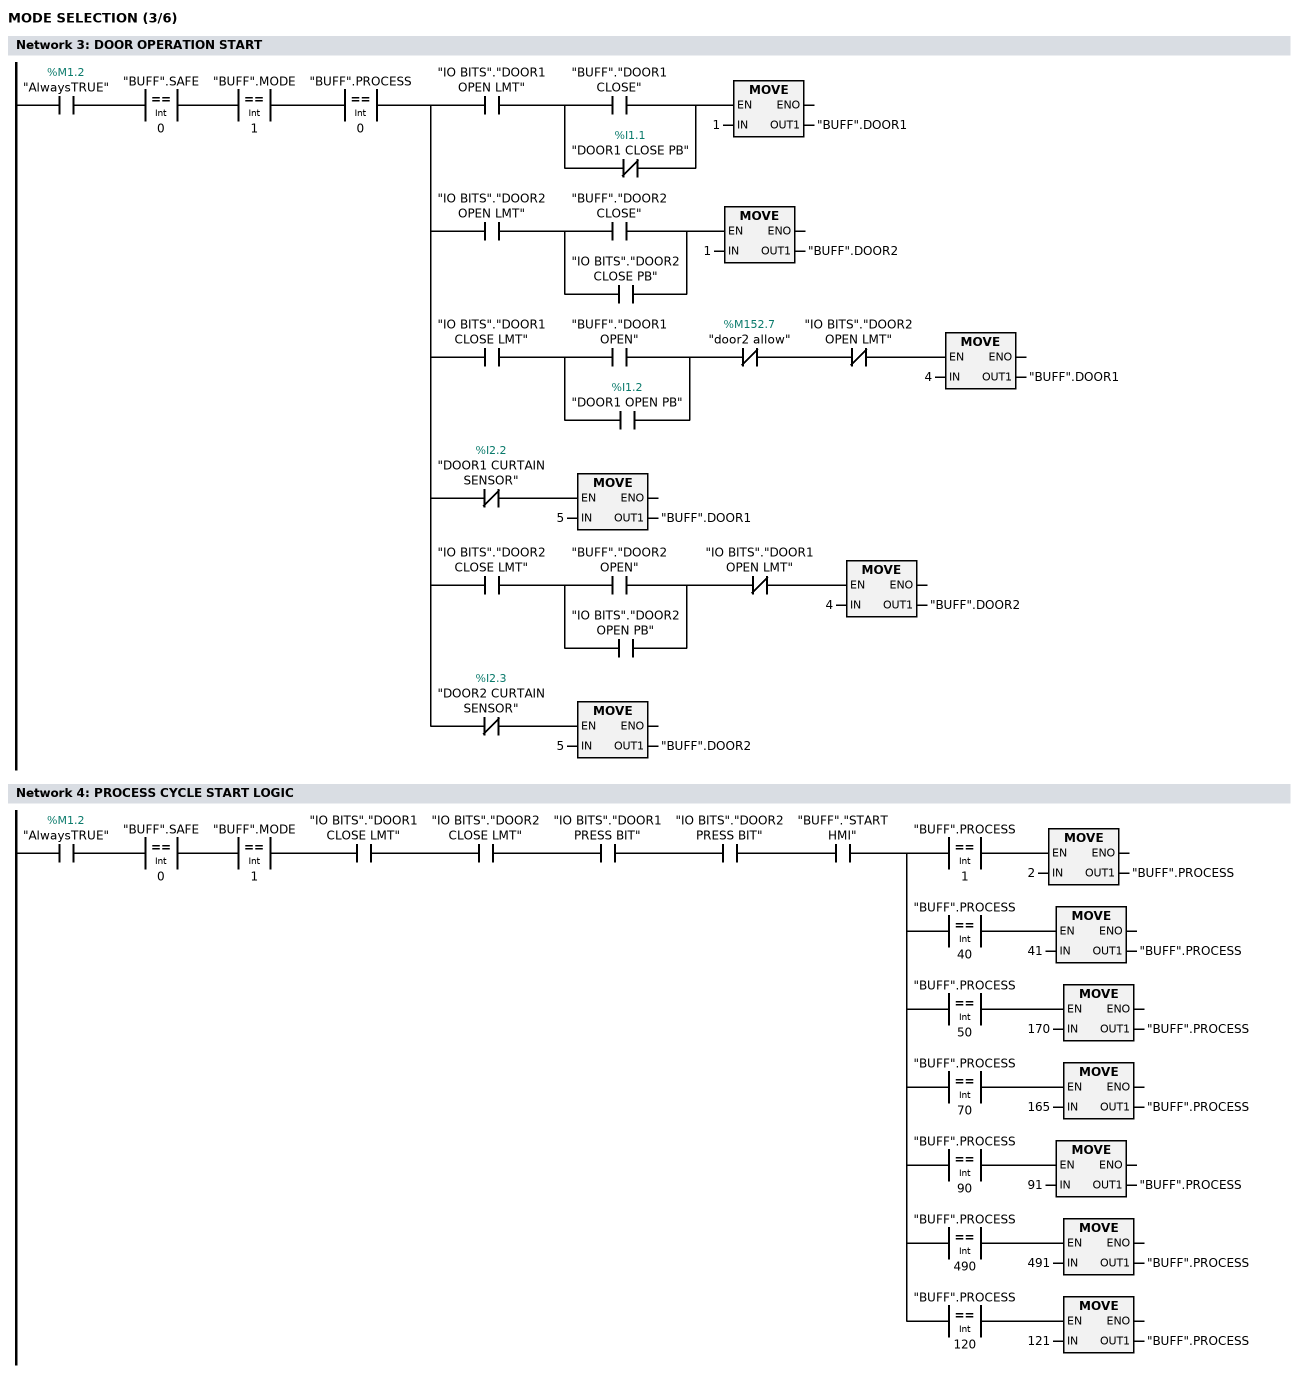
   RUNG wire#powerrail
      Contact( "AlwaysTRUE" )
      { S7_Templates := "SrcType := Int" } EQ_Contact(in1 := "BUFF".SAFE, in2 := 0)
      { S7_Templates := "SrcType := Int" } EQ_Contact(in1 := "BUFF".MODE, in2 := 1)
      { S7_Templates := "SrcType := Int" } EQ_Contact(in1 := "BUFF".PROCESS, in2 := 0)
      wire#w1
      Contact( "IO BITS"."DOOR1 OPEN LMT" )
      wire#w2
      Contact( "BUFF"."DOOR1 CLOSE" )
      wire#w3
      Move(in := 1, out1 => "BUFF".DOOR1)
   END_RUNG
   RUNG wire#w2
      I_Contact( "DOOR1 CLOSE PB" )
   END_RUNG wire#w3
   RUNG wire#w1
      Contact( "IO BITS"."DOOR2 OPEN LMT" )
      wire#w4
      Contact( "BUFF"."DOOR2 CLOSE" )
      wire#w5
      Move(in := 1, out1 => "BUFF".DOOR2)
   END_RUNG
   RUNG wire#w4
      Contact( "IO BITS"."DOOR2 CLOSE PB" )
   END_RUNG wire#w5
   RUNG wire#w1
      Contact( "IO BITS"."DOOR1 CLOSE LMT" )
      wire#w6
      Contact( "BUFF"."DOOR1 OPEN" )
      wire#w7
      I_Contact( "door2 allow" )
      I_Contact( "IO BITS"."DOOR2 OPEN LMT" )
      Move(in := 4, out1 => "BUFF".DOOR1)
   END_RUNG
   RUNG wire#w6
      Contact( "DOOR1 OPEN PB" )
   END_RUNG wire#w7
   RUNG wire#w1
      I_Contact( "DOOR1 CURTAIN SENSOR" )
      Move(in := 5, out1 => "BUFF".DOOR1)
   END_RUNG
   RUNG wire#w1
      Contact( "IO BITS"."DOOR2 CLOSE LMT" )
      wire#w8
      Contact( "BUFF"."DOOR2 OPEN" )
      wire#w9
      I_Contact( "IO BITS"."DOOR1 OPEN LMT" )
      Move(in := 4, out1 => "BUFF".DOOR2)
   END_RUNG
   RUNG wire#w8
      Contact( "IO BITS"."DOOR2 OPEN PB" )
   END_RUNG wire#w9
   RUNG wire#w1
      I_Contact( "DOOR2 CURTAIN SENSOR" )
      Move(in := 5, out1 => "BUFF".DOOR2)
   END_RUNG
   // the same network as SCL:
   #_w1 := "AlwaysTRUE" AND ("BUFF".SAFE = 0) AND ("BUFF".MODE = 1) AND ("BUFF".PROCESS = 0);
   IF #_w1 AND "IO BITS"."DOOR1 OPEN LMT" AND ("BUFF"."DOOR1 CLOSE" OR NOT "DOOR1 CLOSE PB") THEN
       "BUFF".DOOR1 := 1;
   END_IF;
   IF #_w1 AND "IO BITS"."DOOR2 OPEN LMT" AND ("BUFF"."DOOR2 CLOSE" OR "IO BITS"."DOOR2 CLOSE PB") THEN
       "BUFF".DOOR2 := 1;
   END_IF;
   IF #_w1 AND "IO BITS"."DOOR1 CLOSE LMT" AND ("BUFF"."DOOR1 OPEN" OR "DOOR1 OPEN PB") AND NOT "door2 allow" AND NOT "IO BITS"."DOOR2 OPEN LMT" THEN
       "BUFF".DOOR1 := 4;
   END_IF;
   IF #_w1 AND NOT "DOOR1 CURTAIN SENSOR" THEN "BUFF".DOOR1 := 5; END_IF;
   IF #_w1 AND "IO BITS"."DOOR2 CLOSE LMT" AND ("BUFF"."DOOR2 OPEN" OR "IO BITS"."DOOR2 OPEN PB") AND NOT "IO BITS"."DOOR1 OPEN LMT" THEN
       "BUFF".DOOR2 := 4;
   END_IF;
   IF #_w1 AND NOT "DOOR2 CURTAIN SENSOR" THEN "BUFF".DOOR2 := 5; END_IF;
END_REGION

REGION Network 4: PROCESS CYCLE START LOGIC
   RUNG wire#powerrail
      Contact( "AlwaysTRUE" )
      { S7_Templates := "SrcType := Int" } EQ_Contact(in1 := "BUFF".SAFE, in2 := 0)
      { S7_Templates := "SrcType := Int" } EQ_Contact(in1 := "BUFF".MODE, in2 := 1)
      Contact( "IO BITS"."DOOR1 CLOSE LMT" )
      Contact( "IO BITS"."DOOR2 CLOSE LMT" )
      Contact( "IO BITS"."DOOR1 PRESS BIT" )
      Contact( "IO BITS"."DOOR2 PRESS BIT" )
      Contact( "BUFF"."START HMI" )
      wire#w1
      { S7_Templates := "SrcType := Int" } EQ_Contact(in1 := "BUFF".PROCESS, in2 := 1)
      Move(in := 2, out1 => "BUFF".PROCESS)
   END_RUNG
   RUNG wire#w1
      { S7_Templates := "SrcType := Int" } EQ_Contact(in1 := "BUFF".PROCESS, in2 := 40)
      Move(in := 41, out1 => "BUFF".PROCESS)
   END_RUNG
   RUNG wire#w1
      { S7_Templates := "SrcType := Int" } EQ_Contact(in1 := "BUFF".PROCESS, in2 := 50)
      Move(in := 170, out1 => "BUFF".PROCESS)
   END_RUNG
   RUNG wire#w1
      { S7_Templates := "SrcType := Int" } EQ_Contact(in1 := "BUFF".PROCESS, in2 := 70)
      Move(in := 165, out1 => "BUFF".PROCESS)
   END_RUNG
   RUNG wire#w1
      { S7_Templates := "SrcType := Int" } EQ_Contact(in1 := "BUFF".PROCESS, in2 := 90)
      Move(in := 91, out1 => "BUFF".PROCESS)
   END_RUNG
   RUNG wire#w1
      { S7_Templates := "SrcType := Int" } EQ_Contact(in1 := "BUFF".PROCESS, in2 := 490)
      Move(in := 491, out1 => "BUFF".PROCESS)
   END_RUNG
   RUNG wire#w1
      { S7_Templates := "SrcType := Int" } EQ_Contact(in1 := "BUFF".PROCESS, in2 := 120)
      Move(in := 121, out1 => "BUFF".PROCESS)
   END_RUNG
   // the same network as SCL:
   #_w1 := "AlwaysTRUE" AND ("BUFF".SAFE = 0) AND ("BUFF".MODE = 1) AND "IO BITS"."DOOR1 CLOSE LMT" AND "IO BITS"."DOOR2 CLOSE LMT" AND "IO BITS"."DOOR1 PRESS BIT" AND "IO BITS"."DOOR2 PRESS BIT" AND "BUFF"."START HMI";
   IF #_w1 AND ("BUFF".PROCESS = 1) THEN "BUFF".PROCESS := 2; END_IF;
   IF #_w1 AND ("BUFF".PROCESS = 40) THEN "BUFF".PROCESS := 41; END_IF;
   IF #_w1 AND ("BUFF".PROCESS = 50) THEN "BUFF".PROCESS := 170; END_IF;
   IF #_w1 AND ("BUFF".PROCESS = 70) THEN "BUFF".PROCESS := 165; END_IF;
   IF #_w1 AND ("BUFF".PROCESS = 90) THEN "BUFF".PROCESS := 91; END_IF;
   IF #_w1 AND ("BUFF".PROCESS = 490) THEN "BUFF".PROCESS := 491; END_IF;
   IF #_w1 AND ("BUFF".PROCESS = 120) THEN "BUFF".PROCESS := 121; END_IF;
END_REGION

REGION Network 5: DOOR CLOSE LOGIC
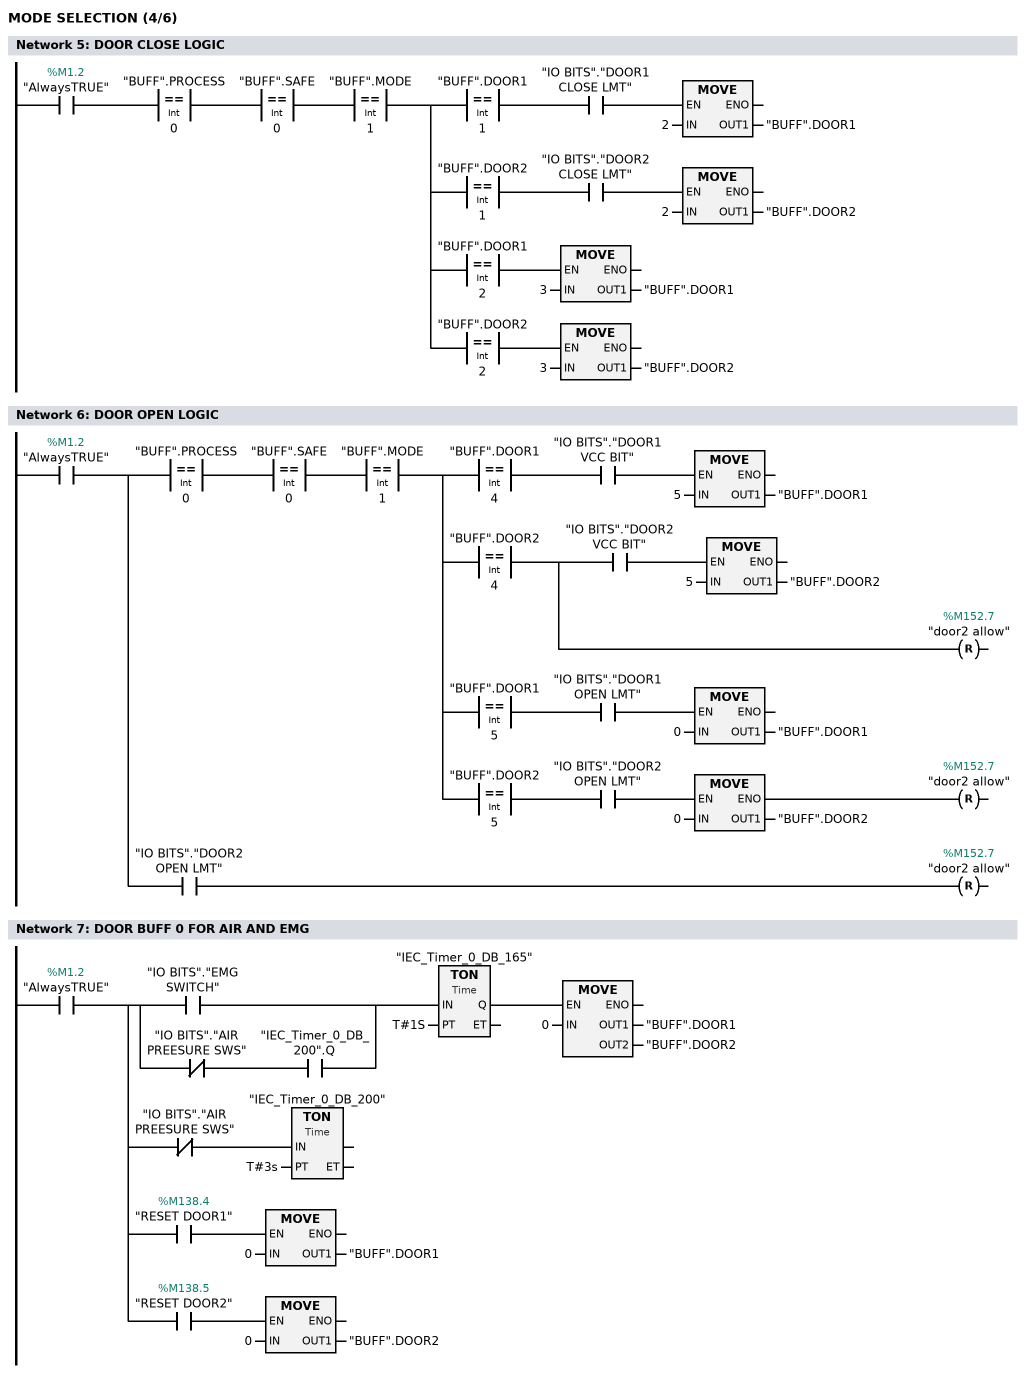
   RUNG wire#powerrail
      Contact( "AlwaysTRUE" )
      { S7_Templates := "SrcType := Int" } EQ_Contact(in1 := "BUFF".PROCESS, in2 := 0)
      { S7_Templates := "SrcType := Int" } EQ_Contact(in1 := "BUFF".SAFE, in2 := 0)
      { S7_Templates := "SrcType := Int" } EQ_Contact(in1 := "BUFF".MODE, in2 := 1)
      wire#w1
      { S7_Templates := "SrcType := Int" } EQ_Contact(in1 := "BUFF".DOOR1, in2 := 1)
      Contact( "IO BITS"."DOOR1 CLOSE LMT" )
      Move(in := 2, out1 => "BUFF".DOOR1)
   END_RUNG
   RUNG wire#w1
      { S7_Templates := "SrcType := Int" } EQ_Contact(in1 := "BUFF".DOOR2, in2 := 1)
      Contact( "IO BITS"."DOOR2 CLOSE LMT" )
      Move(in := 2, out1 => "BUFF".DOOR2)
   END_RUNG
   RUNG wire#w1
      { S7_Templates := "SrcType := Int" } EQ_Contact(in1 := "BUFF".DOOR1, in2 := 2)
      Move(in := 3, out1 => "BUFF".DOOR1)
   END_RUNG
   RUNG wire#w1
      { S7_Templates := "SrcType := Int" } EQ_Contact(in1 := "BUFF".DOOR2, in2 := 2)
      Move(in := 3, out1 => "BUFF".DOOR2)
   END_RUNG
   // the same network as SCL:
   #_w1 := "AlwaysTRUE" AND ("BUFF".PROCESS = 0) AND ("BUFF".SAFE = 0) AND ("BUFF".MODE = 1);
   IF #_w1 AND ("BUFF".DOOR1 = 1) AND "IO BITS"."DOOR1 CLOSE LMT" THEN "BUFF".DOOR1 := 2; END_IF;
   IF #_w1 AND ("BUFF".DOOR2 = 1) AND "IO BITS"."DOOR2 CLOSE LMT" THEN "BUFF".DOOR2 := 2; END_IF;
   IF #_w1 AND ("BUFF".DOOR1 = 2) THEN "BUFF".DOOR1 := 3; END_IF;
   IF #_w1 AND ("BUFF".DOOR2 = 2) THEN "BUFF".DOOR2 := 3; END_IF;
END_REGION

REGION Network 6: DOOR OPEN LOGIC
   RUNG wire#powerrail
      Contact( "AlwaysTRUE" )
      wire#w1
      { S7_Templates := "SrcType := Int" } EQ_Contact(in1 := "BUFF".PROCESS, in2 := 0)
      { S7_Templates := "SrcType := Int" } EQ_Contact(in1 := "BUFF".SAFE, in2 := 0)
      { S7_Templates := "SrcType := Int" } EQ_Contact(in1 := "BUFF".MODE, in2 := 1)
      wire#w2
      { S7_Templates := "SrcType := Int" } EQ_Contact(in1 := "BUFF".DOOR1, in2 := 4)
      Contact( "IO BITS"."DOOR1 VCC BIT" )
      Move(in := 5, out1 => "BUFF".DOOR1)
   END_RUNG
   RUNG wire#w2
      { S7_Templates := "SrcType := Int" } EQ_Contact(in1 := "BUFF".DOOR2, in2 := 4)
      wire#w3
      Contact( "IO BITS"."DOOR2 VCC BIT" )
      Move(in := 5, out1 => "BUFF".DOOR2)
   END_RUNG
   RUNG wire#w3
      R_Coil( "door2 allow" )
   END_RUNG
   RUNG wire#w2
      { S7_Templates := "SrcType := Int" } EQ_Contact(in1 := "BUFF".DOOR1, in2 := 5)
      Contact( "IO BITS"."DOOR1 OPEN LMT" )
      Move(in := 0, out1 => "BUFF".DOOR1)
   END_RUNG
   RUNG wire#w2
      { S7_Templates := "SrcType := Int" } EQ_Contact(in1 := "BUFF".DOOR2, in2 := 5)
      Contact( "IO BITS"."DOOR2 OPEN LMT" )
      Move(in := 0, out1 => "BUFF".DOOR2)
      R_Coil( "door2 allow" )
   END_RUNG
   RUNG wire#w1
      Contact( "IO BITS"."DOOR2 OPEN LMT" )
      R_Coil( "door2 allow" )
   END_RUNG
   // the same network as SCL:
   #_w1 := "AlwaysTRUE" AND ("BUFF".PROCESS = 0) AND ("BUFF".SAFE = 0) AND ("BUFF".MODE = 1);
   IF #_w1 AND ("BUFF".DOOR1 = 4) AND "IO BITS"."DOOR1 VCC BIT" THEN "BUFF".DOOR1 := 5; END_IF;
   #_w2 := #_w1 AND ("BUFF".DOOR2 = 4);
   IF #_w2 AND "IO BITS"."DOOR2 VCC BIT" THEN "BUFF".DOOR2 := 5; END_IF;
   IF #_w2 THEN "door2 allow" := FALSE; END_IF;
   IF #_w1 AND ("BUFF".DOOR1 = 5) AND "IO BITS"."DOOR1 OPEN LMT" THEN "BUFF".DOOR1 := 0; END_IF;
   #_w3 := #_w1 AND ("BUFF".DOOR2 = 5) AND "IO BITS"."DOOR2 OPEN LMT";
   IF #_w3 THEN
       "BUFF".DOOR2 := 0;
       "door2 allow" := FALSE;
   END_IF;
   IF "AlwaysTRUE" AND "IO BITS"."DOOR2 OPEN LMT" THEN "door2 allow" := FALSE; END_IF;
END_REGION

REGION Network 7: DOOR BUFF 0 FOR AIR AND EMG
   RUNG wire#powerrail
      Contact( "AlwaysTRUE" )
      wire#w1
      Contact( "IO BITS"."EMG SWITCH" )
      wire#w2
      { S7_Templates := "time_type := Time" } "IEC_Timer_0_DB_165".TON(pt := T#1S, et =>)
      Move(in := 0, out1 => "BUFF".DOOR1, out2 => "BUFF".DOOR2)
   END_RUNG
   RUNG wire#w1
      I_Contact( "IO BITS"."AIR PREESURE SWS" )
      Contact( "IEC_Timer_0_DB_200".Q )
   END_RUNG wire#w2
   RUNG wire#w1
      I_Contact( "IO BITS"."AIR PREESURE SWS" )
      { S7_Templates := "time_type := Time" } "IEC_Timer_0_DB_200".TON(pt := T#3s, et =>)
   END_RUNG
   RUNG wire#w1
      Contact( "RESET DOOR1" )
      Move(in := 0, out1 => "BUFF".DOOR1)
   END_RUNG
   RUNG wire#w1
      Contact( "RESET DOOR2" )
      Move(in := 0, out1 => "BUFF".DOOR2)
   END_RUNG
   // the same network as SCL:
   "IEC_Timer_0_DB_165".TON(IN := "AlwaysTRUE" AND ("IO BITS"."EMG SWITCH" OR (NOT "IO BITS"."AIR PREESURE SWS" AND "IEC_Timer_0_DB_200".Q)),
                           PT := T#1S);
   IF "IEC_Timer_0_DB_165".Q THEN
       "BUFF".DOOR1 := 0;
       "BUFF".DOOR2 := 0;
   END_IF;
   "IEC_Timer_0_DB_200".TON(IN := "AlwaysTRUE" AND NOT "IO BITS"."AIR PREESURE SWS", PT := T#3s);
   IF "AlwaysTRUE" AND "RESET DOOR1" THEN "BUFF".DOOR1 := 0; END_IF;
   IF "AlwaysTRUE" AND "RESET DOOR2" THEN "BUFF".DOOR2 := 0; END_IF;
END_REGION

REGION Network 8: MANUAL RESET
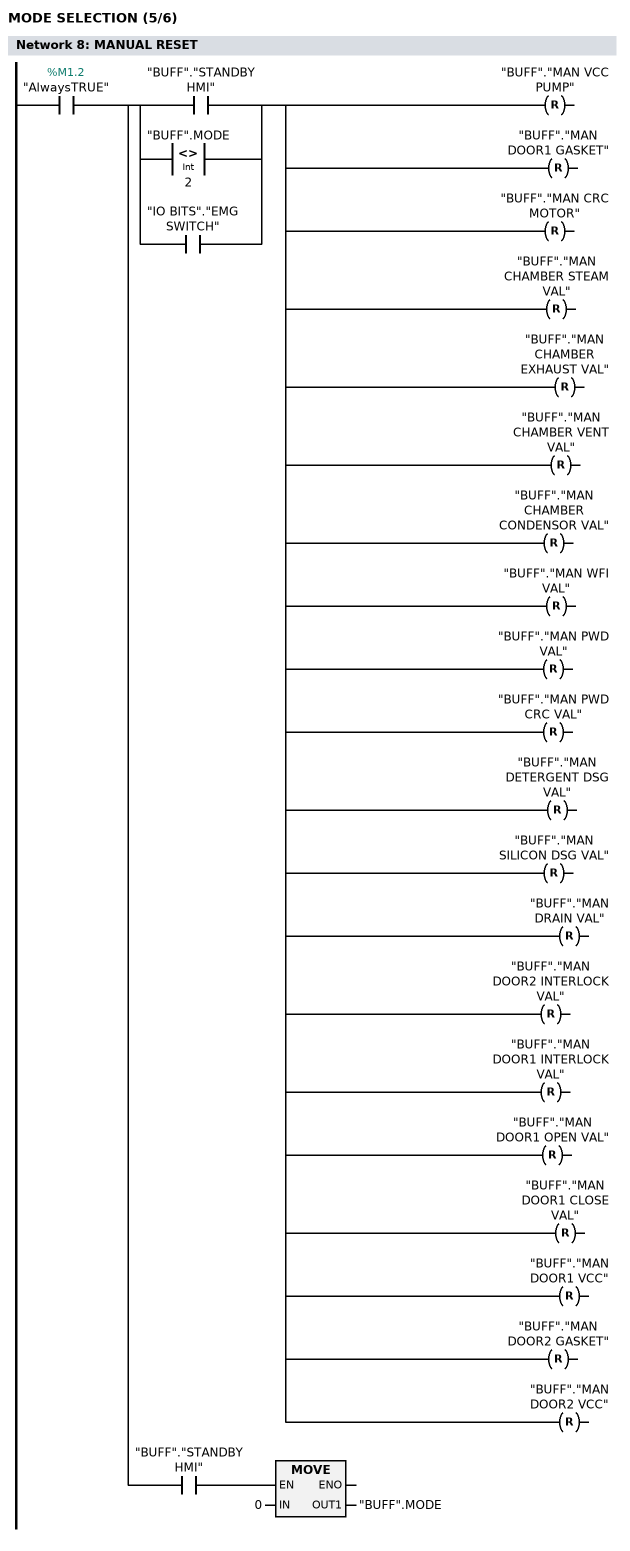
   RUNG wire#powerrail
      Contact( "AlwaysTRUE" )
      wire#w1
      Contact( "BUFF"."STANDBY HMI" )
      wire#w2
      R_Coil( "BUFF"."MAN VCC PUMP" )
   END_RUNG
   RUNG wire#w1
      { S7_Templates := "SrcType := Int" } NE_Contact(in1 := "BUFF".MODE, in2 := 2)
   END_RUNG wire#w2
   RUNG wire#w1
      Contact( "IO BITS"."EMG SWITCH" )
   END_RUNG wire#w2
   RUNG wire#w2
      R_Coil( "BUFF"."MAN DOOR1 GASKET" )
   END_RUNG
   RUNG wire#w2
      R_Coil( "BUFF"."MAN CRC MOTOR" )
   END_RUNG
   RUNG wire#w2
      R_Coil( "BUFF"."MAN CHAMBER STEAM VAL" )
   END_RUNG
   RUNG wire#w2
      R_Coil( "BUFF"."MAN CHAMBER EXHAUST VAL" )
   END_RUNG
   RUNG wire#w2
      R_Coil( "BUFF"."MAN CHAMBER VENT VAL" )
   END_RUNG
   RUNG wire#w2
      R_Coil( "BUFF"."MAN CHAMBER CONDENSOR VAL" )
   END_RUNG
   RUNG wire#w2
      R_Coil( "BUFF"."MAN WFI VAL" )
   END_RUNG
   RUNG wire#w2
      R_Coil( "BUFF"."MAN PWD VAL" )
   END_RUNG
   RUNG wire#w2
      R_Coil( "BUFF"."MAN PWD CRC VAL" )
   END_RUNG
   RUNG wire#w2
      R_Coil( "BUFF"."MAN DETERGENT DSG VAL" )
   END_RUNG
   RUNG wire#w2
      R_Coil( "BUFF"."MAN SILICON DSG VAL" )
   END_RUNG
   RUNG wire#w2
      R_Coil( "BUFF"."MAN DRAIN VAL" )
   END_RUNG
   RUNG wire#w2
      R_Coil( "BUFF"."MAN DOOR2 INTERLOCK VAL" )
   END_RUNG
   RUNG wire#w2
      R_Coil( "BUFF"."MAN DOOR1 INTERLOCK VAL" )
   END_RUNG
   RUNG wire#w2
      R_Coil( "BUFF"."MAN DOOR1 OPEN VAL" )
   END_RUNG
   RUNG wire#w2
      R_Coil( "BUFF"."MAN DOOR1 CLOSE VAL" )
   END_RUNG
   RUNG wire#w2
      R_Coil( "BUFF"."MAN DOOR1 VCC" )
   END_RUNG
   RUNG wire#w2
      R_Coil( "BUFF"."MAN DOOR2 GASKET" )
   END_RUNG
   RUNG wire#w2
      R_Coil( "BUFF"."MAN DOOR2 VCC" )
   END_RUNG
   RUNG wire#w1
      Contact( "BUFF"."STANDBY HMI" )
      Move(in := 0, out1 => "BUFF".MODE)
   END_RUNG
   // the same network as SCL:
   IF "AlwaysTRUE" AND ("BUFF"."STANDBY HMI" OR ("BUFF".MODE <> 2) OR "IO BITS"."EMG SWITCH") THEN
       "BUFF"."MAN VCC PUMP" := FALSE;
       "BUFF"."MAN DOOR1 GASKET" := FALSE;
       "BUFF"."MAN CRC MOTOR" := FALSE;
       "BUFF"."MAN CHAMBER STEAM VAL" := FALSE;
       "BUFF"."MAN CHAMBER EXHAUST VAL" := FALSE;
       "BUFF"."MAN CHAMBER VENT VAL" := FALSE;
       "BUFF"."MAN CHAMBER CONDENSOR VAL" := FALSE;
       "BUFF"."MAN WFI VAL" := FALSE;
       "BUFF"."MAN PWD VAL" := FALSE;
       "BUFF"."MAN PWD CRC VAL" := FALSE;
       "BUFF"."MAN DETERGENT DSG VAL" := FALSE;
       "BUFF"."MAN SILICON DSG VAL" := FALSE;
       "BUFF"."MAN DRAIN VAL" := FALSE;
       "BUFF"."MAN DOOR2 INTERLOCK VAL" := FALSE;
       "BUFF"."MAN DOOR1 INTERLOCK VAL" := FALSE;
       "BUFF"."MAN DOOR1 OPEN VAL" := FALSE;
       "BUFF"."MAN DOOR1 CLOSE VAL" := FALSE;
       "BUFF"."MAN DOOR1 VCC" := FALSE;
       "BUFF"."MAN DOOR2 GASKET" := FALSE;
       "BUFF"."MAN DOOR2 VCC" := FALSE;
   END_IF;
   IF "AlwaysTRUE" AND "BUFF"."STANDBY HMI" THEN "BUFF".MODE := 0; END_IF;
END_REGION

REGION Network 9
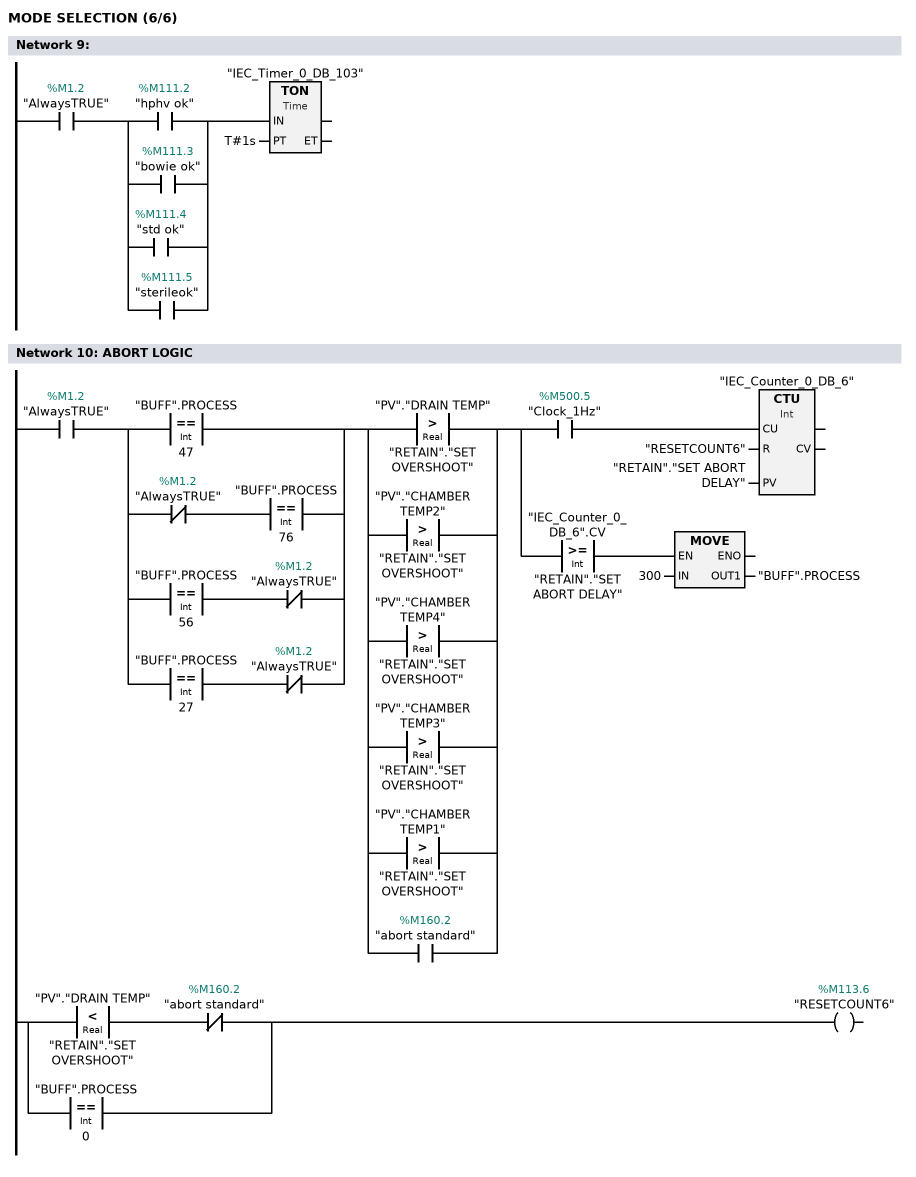
   RUNG wire#powerrail
      Contact( "AlwaysTRUE" )
      wire#w1
      Contact( "hphv ok" )
      wire#w2
      { S7_Templates := "time_type := Time" } "IEC_Timer_0_DB_103".TON(pt := T#1s, et =>)
   END_RUNG
   RUNG wire#w1
      Contact( "bowie ok" )
   END_RUNG wire#w2
   RUNG wire#w1
      Contact( "std ok" )
   END_RUNG wire#w2
   RUNG wire#w1
      Contact( "sterileok" )
   END_RUNG wire#w2
   // the same network as SCL:
   "IEC_Timer_0_DB_103".TON(IN := "AlwaysTRUE" AND ("hphv ok" OR "bowie ok" OR "std ok" OR "sterileok"),
                           PT := T#1s);
END_REGION

REGION Network 10: ABORT LOGIC
   RUNG wire#powerrail
      Contact( "AlwaysTRUE" )
      wire#w1
      { S7_Templates := "SrcType := Int" } EQ_Contact(in1 := "BUFF".PROCESS, in2 := 47)
      wire#w2
      { S7_Templates := "SrcType := Real" } GT_Contact(in1 := "PV"."DRAIN TEMP", in2 := "RETAIN"."SET OVERSHOOT")
      wire#w3
      Contact( "Clock_1Hz" )
      { S7_Templates := "value_type := Int" } "IEC_Counter_0_DB_6".CTU(r := "RESETCOUNT6", pv := "RETAIN"."SET ABORT DELAY", cv =>)
   END_RUNG
   RUNG wire#w1
      I_Contact( "AlwaysTRUE" )
      { S7_Templates := "SrcType := Int" } EQ_Contact(in1 := "BUFF".PROCESS, in2 := 76)
   END_RUNG wire#w2
   RUNG wire#w1
      { S7_Templates := "SrcType := Int" } EQ_Contact(in1 := "BUFF".PROCESS, in2 := 56)
      I_Contact( "AlwaysTRUE" )
   END_RUNG wire#w2
   RUNG wire#w1
      { S7_Templates := "SrcType := Int" } EQ_Contact(in1 := "BUFF".PROCESS, in2 := 27)
      I_Contact( "AlwaysTRUE" )
   END_RUNG wire#w2
   RUNG wire#w2
      { S7_Templates := "SrcType := Real" } GT_Contact(in1 := "PV"."CHAMBER TEMP2", in2 := "RETAIN"."SET OVERSHOOT")
   END_RUNG wire#w3
   RUNG wire#w2
      { S7_Templates := "SrcType := Real" } GT_Contact(in1 := "PV"."CHAMBER TEMP4", in2 := "RETAIN"."SET OVERSHOOT")
   END_RUNG wire#w3
   RUNG wire#w2
      { S7_Templates := "SrcType := Real" } GT_Contact(in1 := "PV"."CHAMBER TEMP3", in2 := "RETAIN"."SET OVERSHOOT")
   END_RUNG wire#w3
   RUNG wire#w2
      { S7_Templates := "SrcType := Real" } GT_Contact(in1 := "PV"."CHAMBER TEMP1", in2 := "RETAIN"."SET OVERSHOOT")
   END_RUNG wire#w3
   RUNG wire#w2
      Contact( "abort standard" )
   END_RUNG wire#w3
   RUNG wire#w3
      { S7_Templates := "SrcType := Int" } GE_Contact(in1 := "IEC_Counter_0_DB_6".CV, in2 := "RETAIN"."SET ABORT DELAY")
      Move(in := 300, out1 => "BUFF".PROCESS)
   END_RUNG
   RUNG wire#powerrail
      { S7_Templates := "SrcType := Real" } LT_Contact(in1 := "PV"."DRAIN TEMP", in2 := "RETAIN"."SET OVERSHOOT")
      I_Contact( "abort standard" )
      wire#w4
      Coil( "RESETCOUNT6" )
   END_RUNG
   RUNG wire#powerrail
      { S7_Templates := "SrcType := Int" } EQ_Contact(in1 := "BUFF".PROCESS, in2 := 0)
   END_RUNG wire#w4
   // the same network as SCL:
   #_w1 := "AlwaysTRUE" AND (("BUFF".PROCESS = 47) OR (NOT "AlwaysTRUE" AND ("BUFF".PROCESS = 76)) OR (("BUFF".PROCESS = 56) AND NOT "AlwaysTRUE") OR (("BUFF".PROCESS = 27) AND NOT "AlwaysTRUE")) AND (("PV"."DRAIN TEMP" > "RETAIN"."SET OVERSHOOT") OR ("PV"."CHAMBER TEMP2" > "RETAIN"."SET OVERSHOOT") OR ("PV"."CHAMBER TEMP4" > "RETAIN"."SET OVERSHOOT") OR ("PV"."CHAMBER TEMP3" > "RETAIN"."SET OVERSHOOT") OR ("PV"."CHAMBER TEMP1" > "RETAIN"."SET OVERSHOOT") OR "abort standard");
   "IEC_Counter_0_DB_6".CTU(CU := #_w1 AND "Clock_1Hz", R := "RESETCOUNT6", PV := "RETAIN"."SET ABORT DELAY");
   IF #_w1 AND ("IEC_Counter_0_DB_6".CV >= "RETAIN"."SET ABORT DELAY") THEN "BUFF".PROCESS := 300; END_IF;
   "RESETCOUNT6" := (("PV"."DRAIN TEMP" < "RETAIN"."SET OVERSHOOT") AND NOT "abort standard") OR ("BUFF".PROCESS = 0);
END_REGION
END_FUNCTION

FUNCTION "ANALOG" : Void   // FC9, LAD
{ S7_Optimized_Access := 'TRUE' }
// stored: SetENOAutomatically false
   VAR_TEMP
      DOOR1_P : Real;
      DOOR2_P : Real;
      CHAMBER_P : Real;
      JACKET_P : Real;
      NOM : Real;
      TEMP1 : Real;
   END_VAR
   VAR_TEMP   // added for the SCL form of the ladder/FBD networks
      _w1 : Bool;
      _w2 : Bool;
      _w3 : Bool;
   END_VAR
BEGIN

REGION Network 1: TEMPERATURE RTD
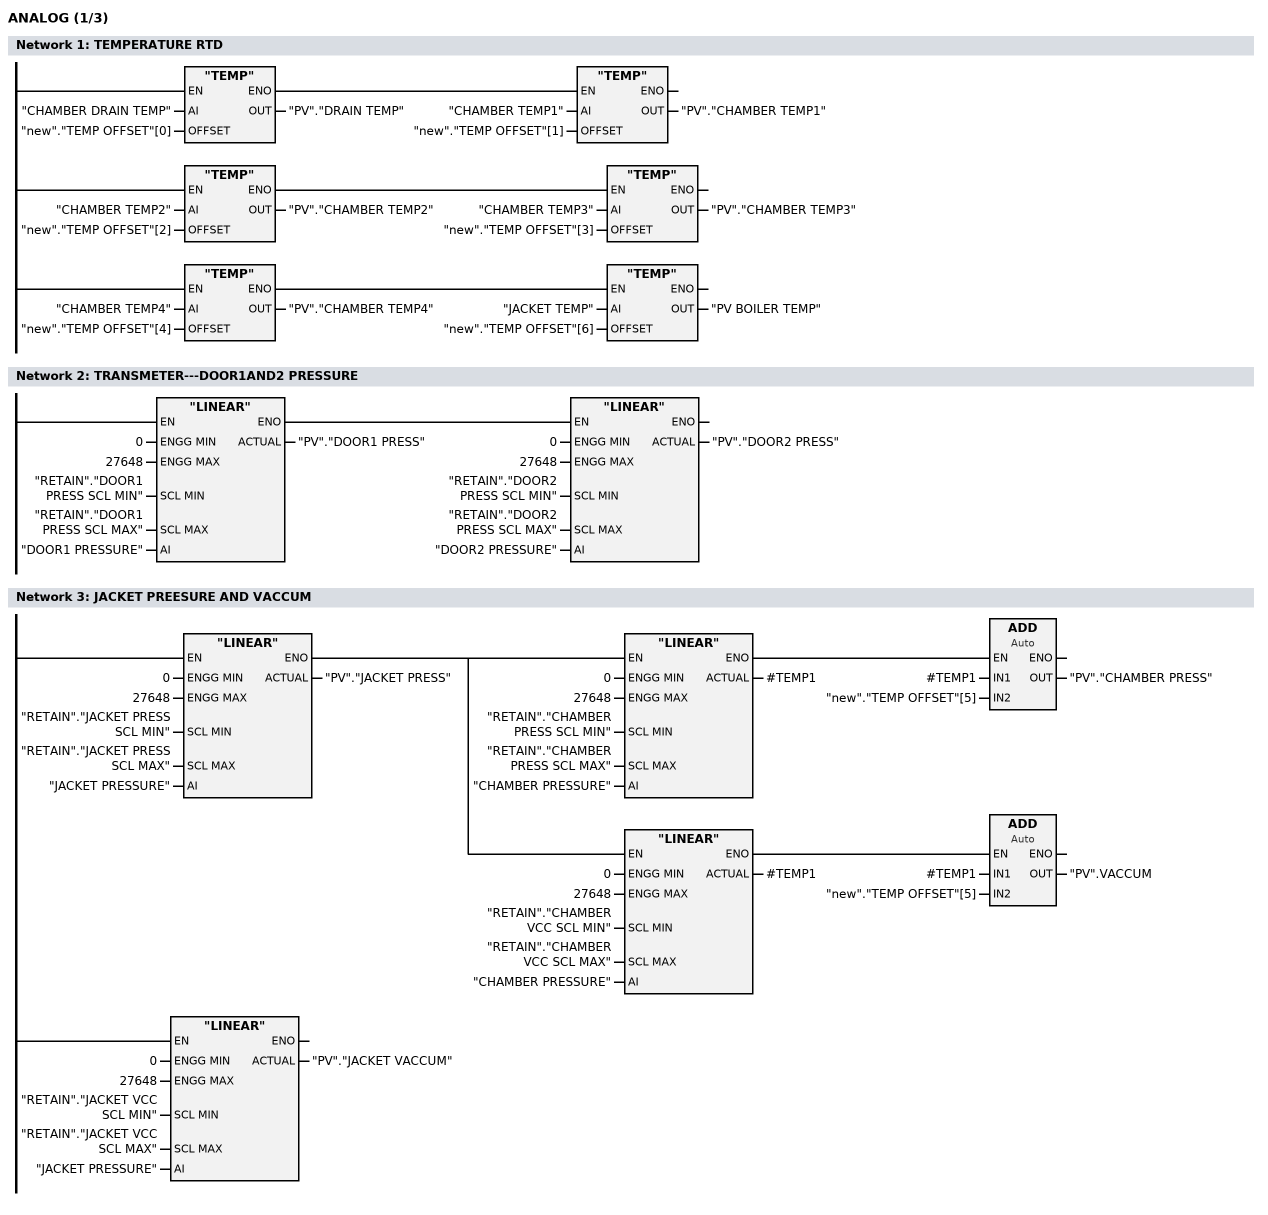
   RUNG wire#powerrail
      "TEMP"(AI := "CHAMBER DRAIN TEMP", OFFSET := "new"."TEMP OFFSET"[0], OUT => "PV"."DRAIN TEMP")
      "TEMP"(AI := "CHAMBER TEMP1", OFFSET := "new"."TEMP OFFSET"[1], OUT => "PV"."CHAMBER TEMP1")
   END_RUNG
   RUNG wire#powerrail
      "TEMP"(AI := "CHAMBER TEMP2", OFFSET := "new"."TEMP OFFSET"[2], OUT => "PV"."CHAMBER TEMP2")
      "TEMP"(AI := "CHAMBER TEMP3", OFFSET := "new"."TEMP OFFSET"[3], OUT => "PV"."CHAMBER TEMP3")
   END_RUNG
   RUNG wire#powerrail
      "TEMP"(AI := "CHAMBER TEMP4", OFFSET := "new"."TEMP OFFSET"[4], OUT => "PV"."CHAMBER TEMP4")
      "TEMP"(AI := "JACKET TEMP", OFFSET := "new"."TEMP OFFSET"[6], OUT => "PV BOILER TEMP")
   END_RUNG
   // the same network as SCL:
   "TEMP"(AI := "CHAMBER DRAIN TEMP", OFFSET := "new"."TEMP OFFSET"[0], OUT => "PV"."DRAIN TEMP", ENO => #_w1);
   IF #_w1 THEN
       "TEMP"(AI := "CHAMBER TEMP1", OFFSET := "new"."TEMP OFFSET"[1], OUT => "PV"."CHAMBER TEMP1");
   END_IF;
   "TEMP"(AI := "CHAMBER TEMP2", OFFSET := "new"."TEMP OFFSET"[2], OUT => "PV"."CHAMBER TEMP2", ENO => #_w2);
   IF #_w2 THEN
       "TEMP"(AI := "CHAMBER TEMP3", OFFSET := "new"."TEMP OFFSET"[3], OUT => "PV"."CHAMBER TEMP3");
   END_IF;
   "TEMP"(AI := "CHAMBER TEMP4", OFFSET := "new"."TEMP OFFSET"[4], OUT => "PV"."CHAMBER TEMP4", ENO => #_w3);
   IF #_w3 THEN
       "TEMP"(AI := "JACKET TEMP", OFFSET := "new"."TEMP OFFSET"[6], OUT => "PV BOILER TEMP");
   END_IF;
END_REGION

REGION Network 2: TRANSMETER---DOOR1AND2 PRESSURE
   RUNG wire#powerrail
      "LINEAR"("ENGG MIN" := 0, "ENGG MAX" := 27648, "SCL MIN" := "RETAIN"."DOOR1 PRESS SCL MIN", "SCL MAX" := "RETAIN"."DOOR1 PRESS SCL MAX", AI := "DOOR1 PRESSURE", ACTUAL => "PV"."DOOR1 PRESS")
      "LINEAR"("ENGG MIN" := 0, "ENGG MAX" := 27648, "SCL MIN" := "RETAIN"."DOOR2 PRESS SCL MIN", "SCL MAX" := "RETAIN"."DOOR2 PRESS SCL MAX", AI := "DOOR2 PRESSURE", ACTUAL => "PV"."DOOR2 PRESS")
   END_RUNG
   // the same network as SCL:
   "LINEAR"("ENGG MIN" := 0,
            "ENGG MAX" := 27648,
            "SCL MIN" := "RETAIN"."DOOR1 PRESS SCL MIN",
            "SCL MAX" := "RETAIN"."DOOR1 PRESS SCL MAX",
            AI := "DOOR1 PRESSURE",
            ACTUAL => "PV"."DOOR1 PRESS",
            ENO => #_w1);
   IF #_w1 THEN
       "LINEAR"("ENGG MIN" := 0,
                "ENGG MAX" := 27648,
                "SCL MIN" := "RETAIN"."DOOR2 PRESS SCL MIN",
                "SCL MAX" := "RETAIN"."DOOR2 PRESS SCL MAX",
                AI := "DOOR2 PRESSURE",
                ACTUAL => "PV"."DOOR2 PRESS");
   END_IF;
END_REGION

REGION Network 3: JACKET PREESURE AND VACCUM
   RUNG wire#powerrail
      "LINEAR"("ENGG MIN" := 0, "ENGG MAX" := 27648, "SCL MIN" := "RETAIN"."JACKET PRESS SCL MIN", "SCL MAX" := "RETAIN"."JACKET PRESS SCL MAX", AI := "JACKET PRESSURE", ACTUAL => "PV"."JACKET PRESS")
      wire#w1
      "LINEAR"("ENGG MIN" := 0, "ENGG MAX" := 27648, "SCL MIN" := "RETAIN"."CHAMBER PRESS SCL MIN", "SCL MAX" := "RETAIN"."CHAMBER PRESS SCL MAX", AI := "CHAMBER PRESSURE", ACTUAL => #TEMP1)
      Add(in1 := #TEMP1, in2 := "new"."TEMP OFFSET"[5], out => "PV"."CHAMBER PRESS")
   END_RUNG
   RUNG wire#w1
      "LINEAR"("ENGG MIN" := 0, "ENGG MAX" := 27648, "SCL MIN" := "RETAIN"."CHAMBER VCC SCL MIN", "SCL MAX" := "RETAIN"."CHAMBER VCC SCL MAX", AI := "CHAMBER PRESSURE", ACTUAL => #TEMP1)
      Add(in1 := #TEMP1, in2 := "new"."TEMP OFFSET"[5], out => "PV".VACCUM)
   END_RUNG
   RUNG wire#powerrail
      "LINEAR"("ENGG MIN" := 0, "ENGG MAX" := 27648, "SCL MIN" := "RETAIN"."JACKET VCC SCL MIN", "SCL MAX" := "RETAIN"."JACKET VCC SCL MAX", AI := "JACKET PRESSURE", ACTUAL => "PV"."JACKET VACCUM")
   END_RUNG
   // the same network as SCL:
   "LINEAR"("ENGG MIN" := 0,
            "ENGG MAX" := 27648,
            "SCL MIN" := "RETAIN"."JACKET PRESS SCL MIN",
            "SCL MAX" := "RETAIN"."JACKET PRESS SCL MAX",
            AI := "JACKET PRESSURE",
            ACTUAL => "PV"."JACKET PRESS",
            ENO => #_w1);
   "LINEAR"(EN := #_w1,
            "ENGG MIN" := 0,
            "ENGG MAX" := 27648,
            "SCL MIN" := "RETAIN"."CHAMBER PRESS SCL MIN",
            "SCL MAX" := "RETAIN"."CHAMBER PRESS SCL MAX",
            AI := "CHAMBER PRESSURE",
            ACTUAL => #TEMP1,
            ENO => #_w2);
   IF #_w2 THEN "PV"."CHAMBER PRESS" := #TEMP1 + "new"."TEMP OFFSET"[5]; END_IF;
   "LINEAR"(EN := #_w1,
            "ENGG MIN" := 0,
            "ENGG MAX" := 27648,
            "SCL MIN" := "RETAIN"."CHAMBER VCC SCL MIN",
            "SCL MAX" := "RETAIN"."CHAMBER VCC SCL MAX",
            AI := "CHAMBER PRESSURE",
            ACTUAL => #TEMP1,
            ENO => #_w3);
   IF #_w3 THEN "PV".VACCUM := #TEMP1 + "new"."TEMP OFFSET"[5]; END_IF;
   "LINEAR"("ENGG MIN" := 0,
            "ENGG MAX" := 27648,
            "SCL MIN" := "RETAIN"."JACKET VCC SCL MIN",
            "SCL MAX" := "RETAIN"."JACKET VCC SCL MAX",
            AI := "JACKET PRESSURE",
            ACTUAL => "PV"."JACKET VACCUM");
END_REGION

REGION Network 4: DOOR1AND 2 VACCUM
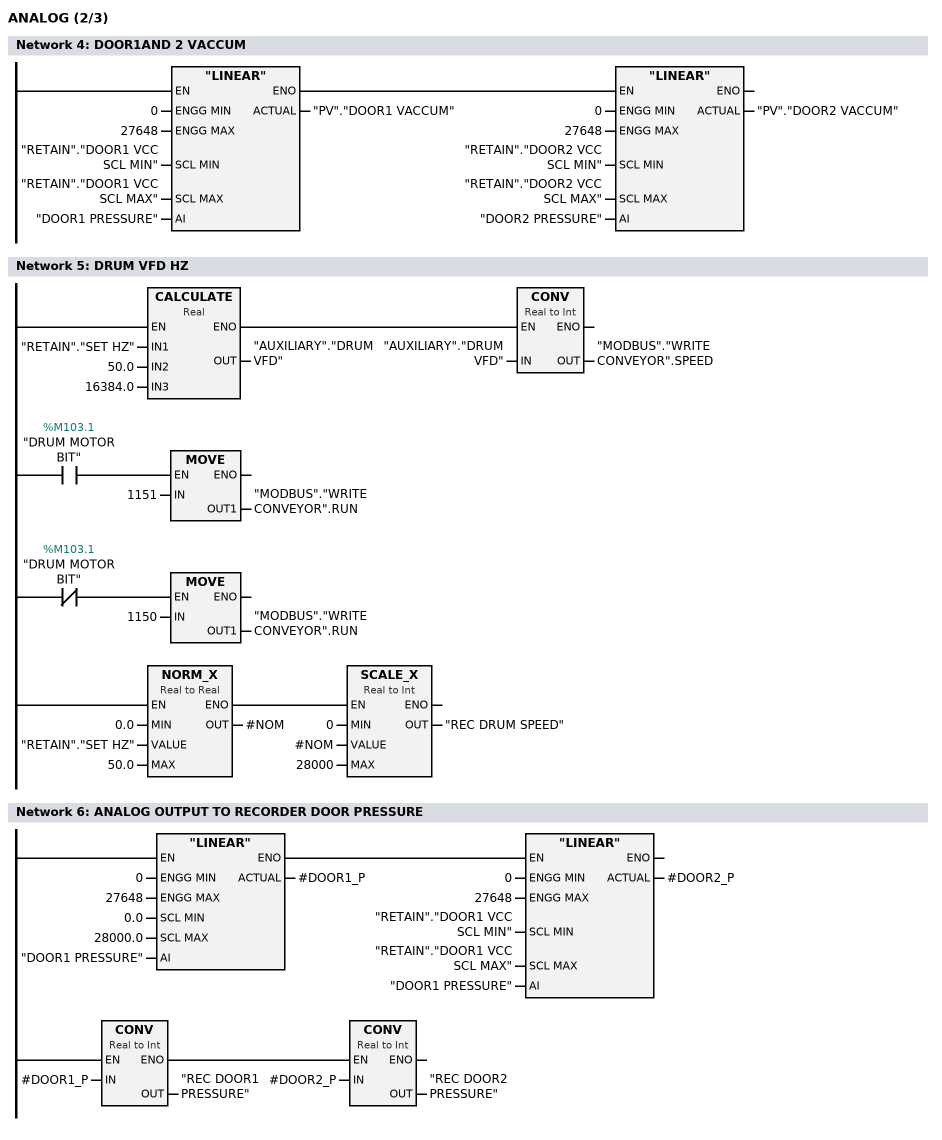
   RUNG wire#powerrail
      "LINEAR"("ENGG MIN" := 0, "ENGG MAX" := 27648, "SCL MIN" := "RETAIN"."DOOR1 VCC SCL MIN", "SCL MAX" := "RETAIN"."DOOR1 VCC SCL MAX", AI := "DOOR1 PRESSURE", ACTUAL => "PV"."DOOR1 VACCUM")
      "LINEAR"("ENGG MIN" := 0, "ENGG MAX" := 27648, "SCL MIN" := "RETAIN"."DOOR2 VCC SCL MIN", "SCL MAX" := "RETAIN"."DOOR2 VCC SCL MAX", AI := "DOOR2 PRESSURE", ACTUAL => "PV"."DOOR2 VACCUM")
   END_RUNG
   // the same network as SCL:
   "LINEAR"("ENGG MIN" := 0,
            "ENGG MAX" := 27648,
            "SCL MIN" := "RETAIN"."DOOR1 VCC SCL MIN",
            "SCL MAX" := "RETAIN"."DOOR1 VCC SCL MAX",
            AI := "DOOR1 PRESSURE",
            ACTUAL => "PV"."DOOR1 VACCUM",
            ENO => #_w1);
   IF #_w1 THEN
       "LINEAR"("ENGG MIN" := 0,
                "ENGG MAX" := 27648,
                "SCL MIN" := "RETAIN"."DOOR2 VCC SCL MIN",
                "SCL MAX" := "RETAIN"."DOOR2 VCC SCL MAX",
                AI := "DOOR2 PRESSURE",
                ACTUAL => "PV"."DOOR2 VACCUM");
   END_IF;
END_REGION

REGION Network 5: DRUM VFD HZ
   RUNG wire#powerrail
      { S7_Templates := "SrcType := Real"; S7_Expression := "(IN1/IN2)*IN3" } Calculate(in1 := "RETAIN"."SET HZ", in2 := 50.0, in3 := 16384.0, out => "AUXILIARY"."DRUM VFD")
      { S7_Templates := "[SrcType := Real, DestType := Int]" } Convert(in := "AUXILIARY"."DRUM VFD", out => "MODBUS"."WRITE CONVEYOR".SPEED)
   END_RUNG
   RUNG wire#powerrail
      Contact( "DRUM MOTOR BIT" )
      Move(in := 1151, out1 => "MODBUS"."WRITE CONVEYOR".RUN)
   END_RUNG
   RUNG wire#powerrail
      I_Contact( "DRUM MOTOR BIT" )
      Move(in := 1150, out1 => "MODBUS"."WRITE CONVEYOR".RUN)
   END_RUNG
   RUNG wire#powerrail
      { S7_Templates := "[SrcType := Real, DestType := Real]" } Normalize(min := 0.0, value := "RETAIN"."SET HZ", max := 50.0, out => #NOM)
      { S7_Templates := "[SrcType := Real, DestType := Int]" } Scale(min := 0, value := #NOM, max := 28000, out => "REC DRUM SPEED")
   END_RUNG
   // the same network as SCL:
   "AUXILIARY"."DRUM VFD" := ("RETAIN"."SET HZ"/50.0)*16384.0;
   "MODBUS"."WRITE CONVEYOR".SPEED := REAL_TO_INT("AUXILIARY"."DRUM VFD");
   IF "DRUM MOTOR BIT" THEN "MODBUS"."WRITE CONVEYOR".RUN := 1151; END_IF;
   IF NOT "DRUM MOTOR BIT" THEN "MODBUS"."WRITE CONVEYOR".RUN := 1150; END_IF;
   #NOM := NORM_X(MIN := 0.0, VALUE := "RETAIN"."SET HZ", MAX := 50.0);
   "REC DRUM SPEED" := SCALE_X(MIN := 0, VALUE := #NOM, MAX := 28000);
END_REGION

REGION Network 6: ANALOG OUTPUT TO RECORDER DOOR PRESSURE
   RUNG wire#powerrail
      "LINEAR"("ENGG MIN" := 0, "ENGG MAX" := 27648, "SCL MIN" := 0.0, "SCL MAX" := 28000.0, AI := "DOOR1 PRESSURE", ACTUAL => #DOOR1_P)
      "LINEAR"("ENGG MIN" := 0, "ENGG MAX" := 27648, "SCL MIN" := "RETAIN"."DOOR1 VCC SCL MIN", "SCL MAX" := "RETAIN"."DOOR1 VCC SCL MAX", AI := "DOOR1 PRESSURE", ACTUAL => #DOOR2_P)
   END_RUNG
   RUNG wire#powerrail
      { S7_Templates := "[SrcType := Real, DestType := Int]" } Convert(in := #DOOR1_P, out => "REC DOOR1 PRESSURE")
      { S7_Templates := "[SrcType := Real, DestType := Int]" } Convert(in := #DOOR2_P, out => "REC DOOR2 PRESSURE")
   END_RUNG
   // the same network as SCL:
   "LINEAR"("ENGG MIN" := 0,
            "ENGG MAX" := 27648,
            "SCL MIN" := 0.0,
            "SCL MAX" := 28000.0,
            AI := "DOOR1 PRESSURE",
            ACTUAL => #DOOR1_P,
            ENO => #_w1);
   IF #_w1 THEN
       "LINEAR"("ENGG MIN" := 0,
                "ENGG MAX" := 27648,
                "SCL MIN" := "RETAIN"."DOOR1 VCC SCL MIN",
                "SCL MAX" := "RETAIN"."DOOR1 VCC SCL MAX",
                AI := "DOOR1 PRESSURE",
                ACTUAL => #DOOR2_P);
   END_IF;
   "REC DOOR1 PRESSURE" := REAL_TO_INT(#DOOR1_P);
   "REC DOOR2 PRESSURE" := REAL_TO_INT(#DOOR2_P);
END_REGION

REGION Network 7: ANALOG OUTPUT TO RECORDER CHAMBER AND JACKET
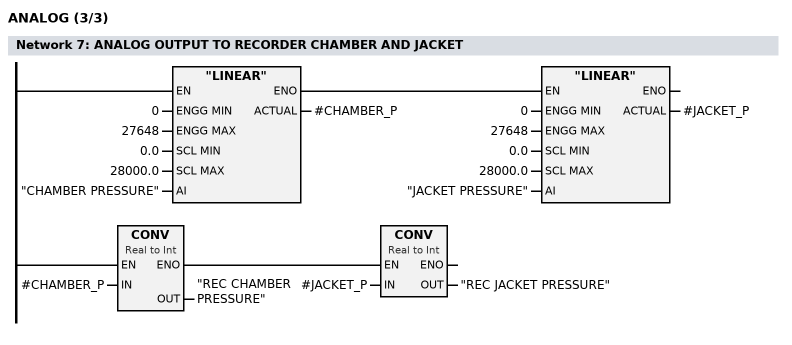
   RUNG wire#powerrail
      "LINEAR"("ENGG MIN" := 0, "ENGG MAX" := 27648, "SCL MIN" := 0.0, "SCL MAX" := 28000.0, AI := "CHAMBER PRESSURE", ACTUAL => #CHAMBER_P)
      "LINEAR"("ENGG MIN" := 0, "ENGG MAX" := 27648, "SCL MIN" := 0.0, "SCL MAX" := 28000.0, AI := "JACKET PRESSURE", ACTUAL => #JACKET_P)
   END_RUNG
   RUNG wire#powerrail
      { S7_Templates := "[SrcType := Real, DestType := Int]" } Convert(in := #CHAMBER_P, out => "REC CHAMBER PRESSURE")
      { S7_Templates := "[SrcType := Real, DestType := Int]" } Convert(in := #JACKET_P, out => "REC JACKET PRESSURE")
   END_RUNG
   // the same network as SCL:
   "LINEAR"("ENGG MIN" := 0,
            "ENGG MAX" := 27648,
            "SCL MIN" := 0.0,
            "SCL MAX" := 28000.0,
            AI := "CHAMBER PRESSURE",
            ACTUAL => #CHAMBER_P,
            ENO => #_w1);
   IF #_w1 THEN
       "LINEAR"("ENGG MIN" := 0,
                "ENGG MAX" := 27648,
                "SCL MIN" := 0.0,
                "SCL MAX" := 28000.0,
                AI := "JACKET PRESSURE",
                ACTUAL => #JACKET_P);
   END_IF;
   "REC CHAMBER PRESSURE" := REAL_TO_INT(#CHAMBER_P);
   "REC JACKET PRESSURE" := REAL_TO_INT(#JACKET_P);
END_REGION
END_FUNCTION

FUNCTION "TEMP" : Void   // FC14, LAD
{ S7_Optimized_Access := 'TRUE' }
// stored: SetENOAutomatically false
   VAR_INPUT
      AI : Int;
      OFFSET : Real;
   END_VAR
   VAR_OUTPUT
      OUT : Real;
   END_VAR
   VAR_TEMP
      TEMP1 : Real;
      temp2 : Real;
   END_VAR
BEGIN

REGION Network 1
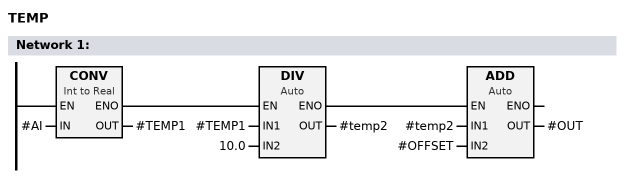
   RUNG wire#powerrail
      { S7_Templates := "[SrcType := Int, DestType := Real]" } Convert(in := #AI, out => #TEMP1)
      Div(in1 := #TEMP1, in2 := 10.0, out => #temp2)
      Add(in1 := #temp2, in2 := #OFFSET, out => #OUT)
   END_RUNG
   // the same network as SCL:
   #TEMP1 := INT_TO_REAL(#AI);
   #temp2 := #TEMP1 / 10.0;
   #OUT := #temp2 + #OFFSET;
END_REGION
END_FUNCTION

FUNCTION "LINEAR" : Void   // FC15, LAD
{ S7_Optimized_Access := 'TRUE' }
// stored: SetENOAutomatically false
   VAR_INPUT
      "ENGG MIN" : Int;
      "ENGG MAX" : Int;
      "SCL MIN" : Real;
      "SCL MAX" : Real;
      AI : Int;
   END_VAR
   VAR_OUTPUT
      ACTUAL : Real;
   END_VAR
   VAR_TEMP
      NOM : Real;
   END_VAR
BEGIN

REGION Network 1
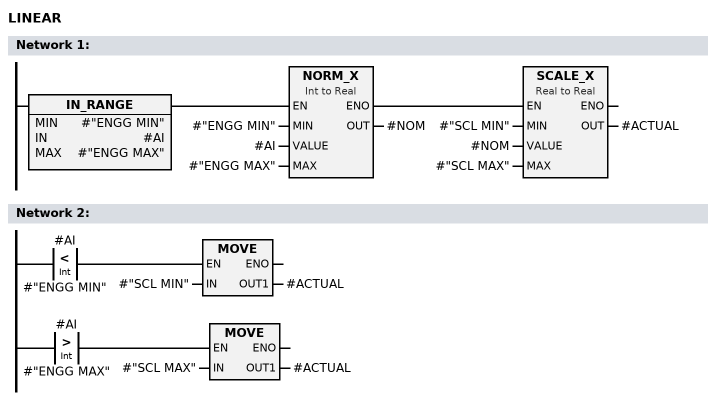
   RUNG wire#powerrail
      { S7_Templates := "SrcType := Int" } InRange(min := #"ENGG MIN", in := #AI, max := #"ENGG MAX")
      { S7_Templates := "[SrcType := Int, DestType := Real]" } Normalize(min := #"ENGG MIN", value := #AI, max := #"ENGG MAX", out => #NOM)
      { S7_Templates := "[SrcType := Real, DestType := Real]" } Scale(min := #"SCL MIN", value := #NOM, max := #"SCL MAX", out => #ACTUAL)
   END_RUNG
   // the same network as SCL:
   IF (#"ENGG MIN" <= #AI) AND (#AI <= #"ENGG MAX") THEN
       #NOM := NORM_X(MIN := #"ENGG MIN", VALUE := #AI, MAX := #"ENGG MAX");
       #ACTUAL := SCALE_X(MIN := #"SCL MIN", VALUE := #NOM, MAX := #"SCL MAX");
   END_IF;
END_REGION

REGION Network 2
   RUNG wire#powerrail
      { S7_Templates := "SrcType := Int" } LT_Contact(in1 := #AI, in2 := #"ENGG MIN")
      Move(in := #"SCL MIN", out1 => #ACTUAL)
   END_RUNG
   RUNG wire#powerrail
      { S7_Templates := "SrcType := Int" } GT_Contact(in1 := #AI, in2 := #"ENGG MAX")
      Move(in := #"SCL MAX", out1 => #ACTUAL)
   END_RUNG
   // the same network as SCL:
   IF #AI < #"ENGG MIN" THEN #ACTUAL := #"SCL MIN"; END_IF;
   IF #AI > #"ENGG MAX" THEN #ACTUAL := #"SCL MAX"; END_IF;
END_REGION
END_FUNCTION

FUNCTION "DELTA" : Void   // FC18, LAD
{ S7_Optimized_Access := 'TRUE' }
// stored: SetENOAutomatically false
   VAR_TEMP
      "F1 VALUE" : Real;
      "F2 VALUE" : Real;
      "F3 VALUE" : Real;
      "F4 VALUE" : Real;
      "F5 VALUE" : Real;
   END_VAR
   VAR_TEMP   // added for the SCL form of the ladder/FBD networks
      _w1 : Bool;
      _w2 : Bool;
      _w3 : Bool;
      _w4 : Bool;
      _w5 : Bool;
      _w6 : Bool;
      _w7 : Bool;
      _w8 : Bool;
      _w9 : Bool;
      _w10 : Bool;
      _w11 : Bool;
      _w12 : Bool;
   END_VAR
BEGIN

REGION Network 1
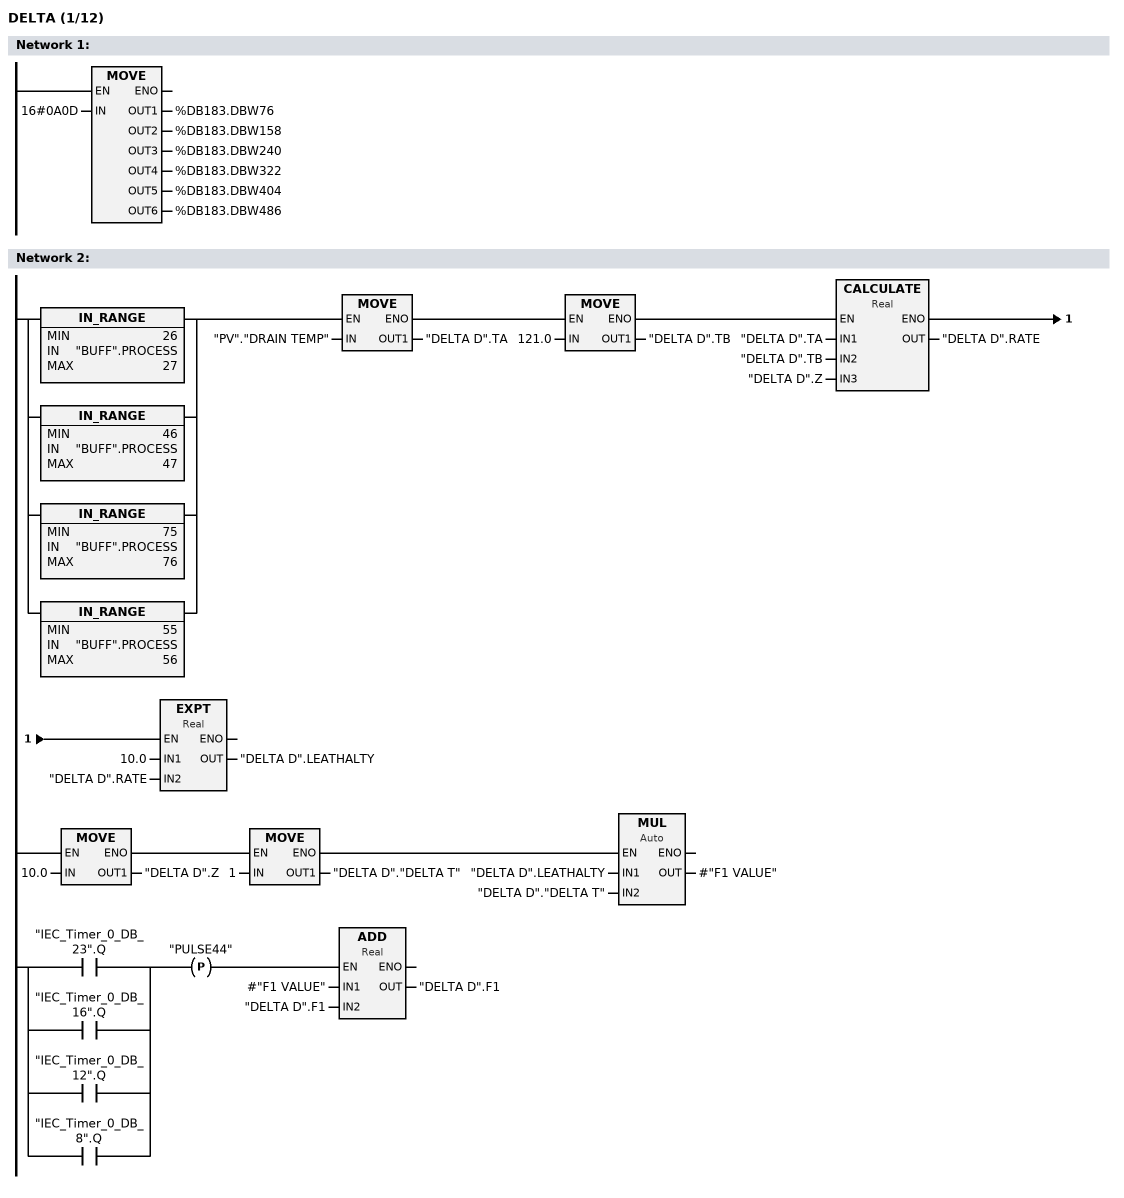
   RUNG wire#powerrail
      Move(in := 16#0A0D, out1 => %DB183.DBW76, out2 => %DB183.DBW158, out3 => %DB183.DBW240, out4 => %DB183.DBW322, out5 => %DB183.DBW404, out6 => %DB183.DBW486)
   END_RUNG
   // the same network as SCL:
   %DB183.DBW76 := 16#0A0D;
   %DB183.DBW158 := 16#0A0D;
   %DB183.DBW240 := 16#0A0D;
   %DB183.DBW322 := 16#0A0D;
   %DB183.DBW404 := 16#0A0D;
   %DB183.DBW486 := 16#0A0D;
END_REGION

REGION Network 2
   IF ((26 <= "BUFF".PROCESS) AND ("BUFF".PROCESS <= 27)) OR ((46 <= "BUFF".PROCESS) AND ("BUFF".PROCESS <= 47)) OR ((75 <= "BUFF".PROCESS) AND ("BUFF".PROCESS <= 76)) OR ((55 <= "BUFF".PROCESS) AND ("BUFF".PROCESS <= 56)) THEN
       "DELTA D".TA := "PV"."DRAIN TEMP";
       "DELTA D".TB := 121.0;
       "DELTA D".RATE := ("DELTA D".TA-"DELTA D".TB)/"DELTA D".Z;
       "DELTA D".LEATHALTY := 10.0 ** "DELTA D".RATE;
   END_IF;
   "DELTA D".Z := 10.0;
   "DELTA D"."DELTA T" := 1;
   #"F1 VALUE" := "DELTA D".LEATHALTY * "DELTA D"."DELTA T";
   #_w1 := "IEC_Timer_0_DB_23".Q OR "IEC_Timer_0_DB_16".Q OR "IEC_Timer_0_DB_12".Q OR "IEC_Timer_0_DB_8".Q;
   #_w2 := #_w1 AND NOT "PULSE44";   // rising edge
   "PULSE44" := #_w1;
   IF #_w2 THEN "DELTA D".F1 := #"F1 VALUE" + "DELTA D".F1; END_IF;
END_REGION

REGION Network 3
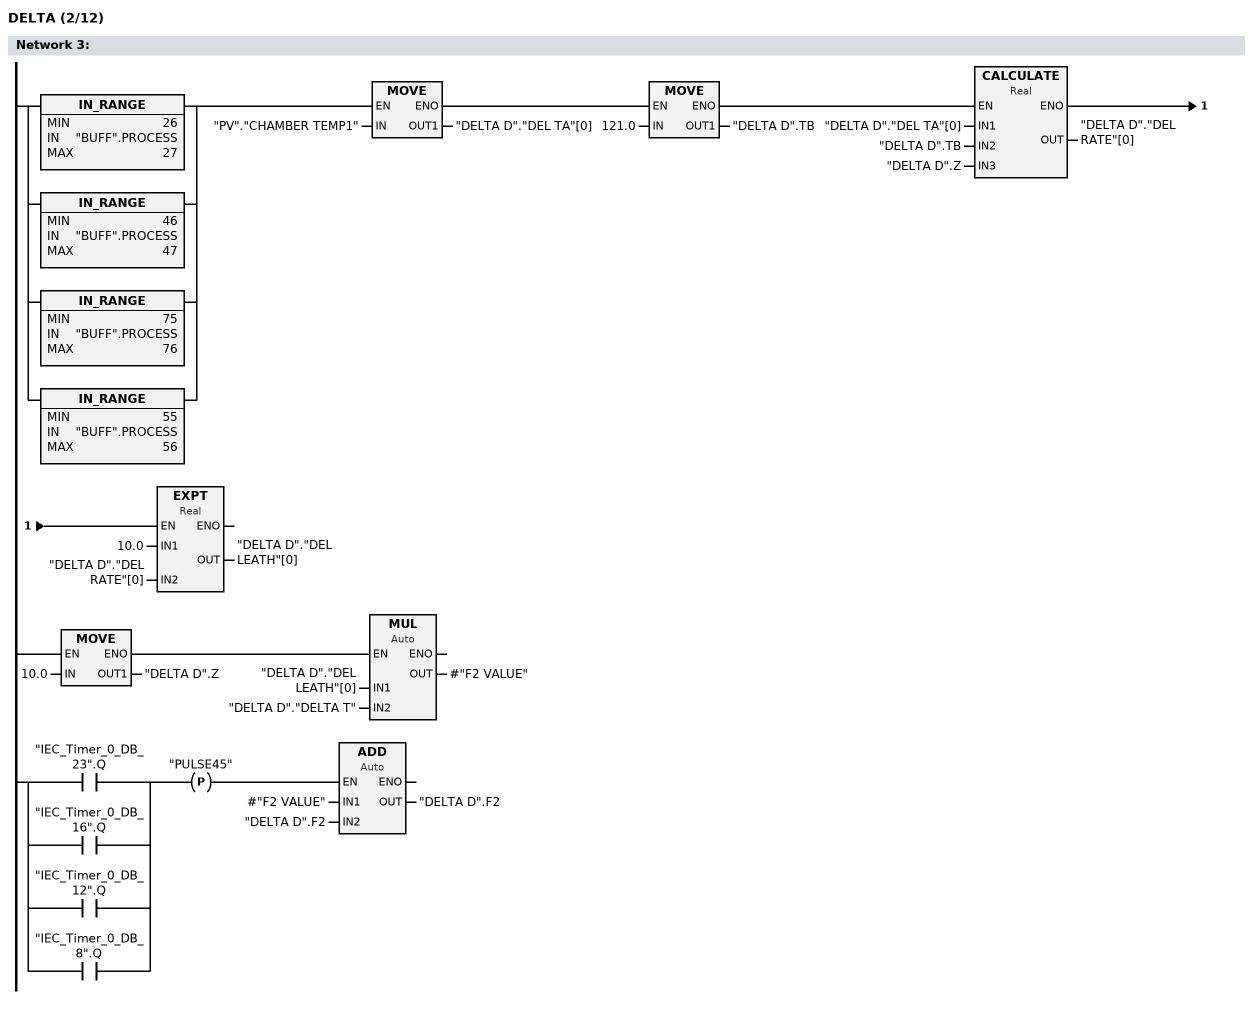
   IF ((26 <= "BUFF".PROCESS) AND ("BUFF".PROCESS <= 27)) OR ((46 <= "BUFF".PROCESS) AND ("BUFF".PROCESS <= 47)) OR ((75 <= "BUFF".PROCESS) AND ("BUFF".PROCESS <= 76)) OR ((55 <= "BUFF".PROCESS) AND ("BUFF".PROCESS <= 56)) THEN
       "DELTA D"."DEL TA"[0] := "PV"."CHAMBER TEMP1";
       "DELTA D".TB := 121.0;
       "DELTA D"."DEL RATE"[0] := ("DELTA D"."DEL TA"[0]-"DELTA D".TB)/"DELTA D".Z;
       "DELTA D"."DEL LEATH"[0] := 10.0 ** "DELTA D"."DEL RATE"[0];
   END_IF;
   "DELTA D".Z := 10.0;
   #"F2 VALUE" := "DELTA D"."DEL LEATH"[0] * "DELTA D"."DELTA T";
   #_w1 := "IEC_Timer_0_DB_23".Q OR "IEC_Timer_0_DB_16".Q OR "IEC_Timer_0_DB_12".Q OR "IEC_Timer_0_DB_8".Q;
   #_w2 := #_w1 AND NOT "PULSE45";   // rising edge
   "PULSE45" := #_w1;
   IF #_w2 THEN "DELTA D".F2 := #"F2 VALUE" + "DELTA D".F2; END_IF;
END_REGION

REGION Network 4
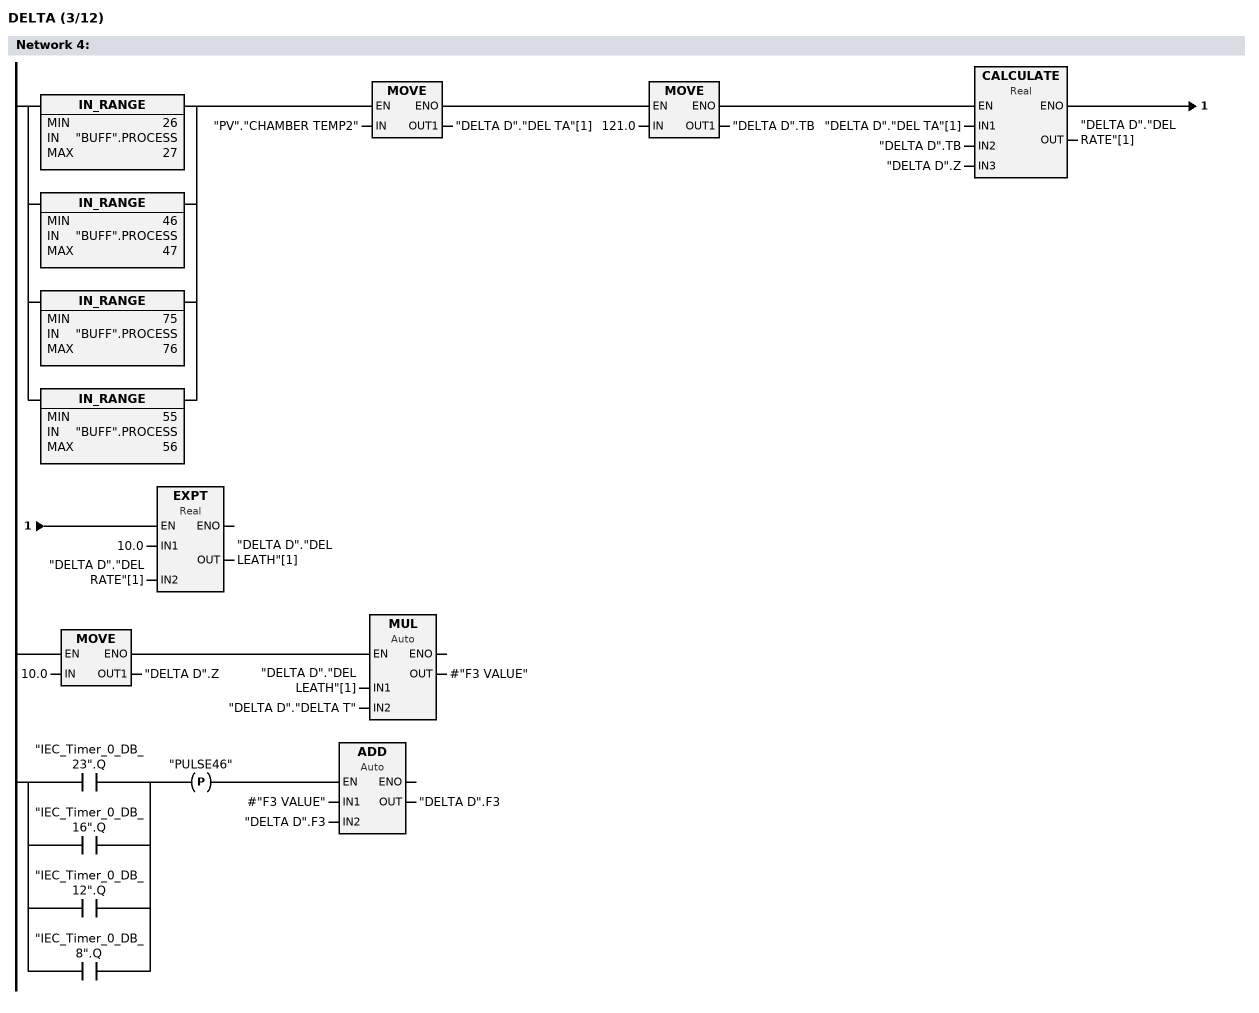
   IF ((26 <= "BUFF".PROCESS) AND ("BUFF".PROCESS <= 27)) OR ((46 <= "BUFF".PROCESS) AND ("BUFF".PROCESS <= 47)) OR ((75 <= "BUFF".PROCESS) AND ("BUFF".PROCESS <= 76)) OR ((55 <= "BUFF".PROCESS) AND ("BUFF".PROCESS <= 56)) THEN
       "DELTA D"."DEL TA"[1] := "PV"."CHAMBER TEMP2";
       "DELTA D".TB := 121.0;
       "DELTA D"."DEL RATE"[1] := ("DELTA D"."DEL TA"[1]-"DELTA D".TB)/"DELTA D".Z;
       "DELTA D"."DEL LEATH"[1] := 10.0 ** "DELTA D"."DEL RATE"[1];
   END_IF;
   "DELTA D".Z := 10.0;
   #"F3 VALUE" := "DELTA D"."DEL LEATH"[1] * "DELTA D"."DELTA T";
   #_w1 := "IEC_Timer_0_DB_23".Q OR "IEC_Timer_0_DB_16".Q OR "IEC_Timer_0_DB_12".Q OR "IEC_Timer_0_DB_8".Q;
   #_w2 := #_w1 AND NOT "PULSE46";   // rising edge
   "PULSE46" := #_w1;
   IF #_w2 THEN "DELTA D".F3 := #"F3 VALUE" + "DELTA D".F3; END_IF;
END_REGION

REGION Network 5
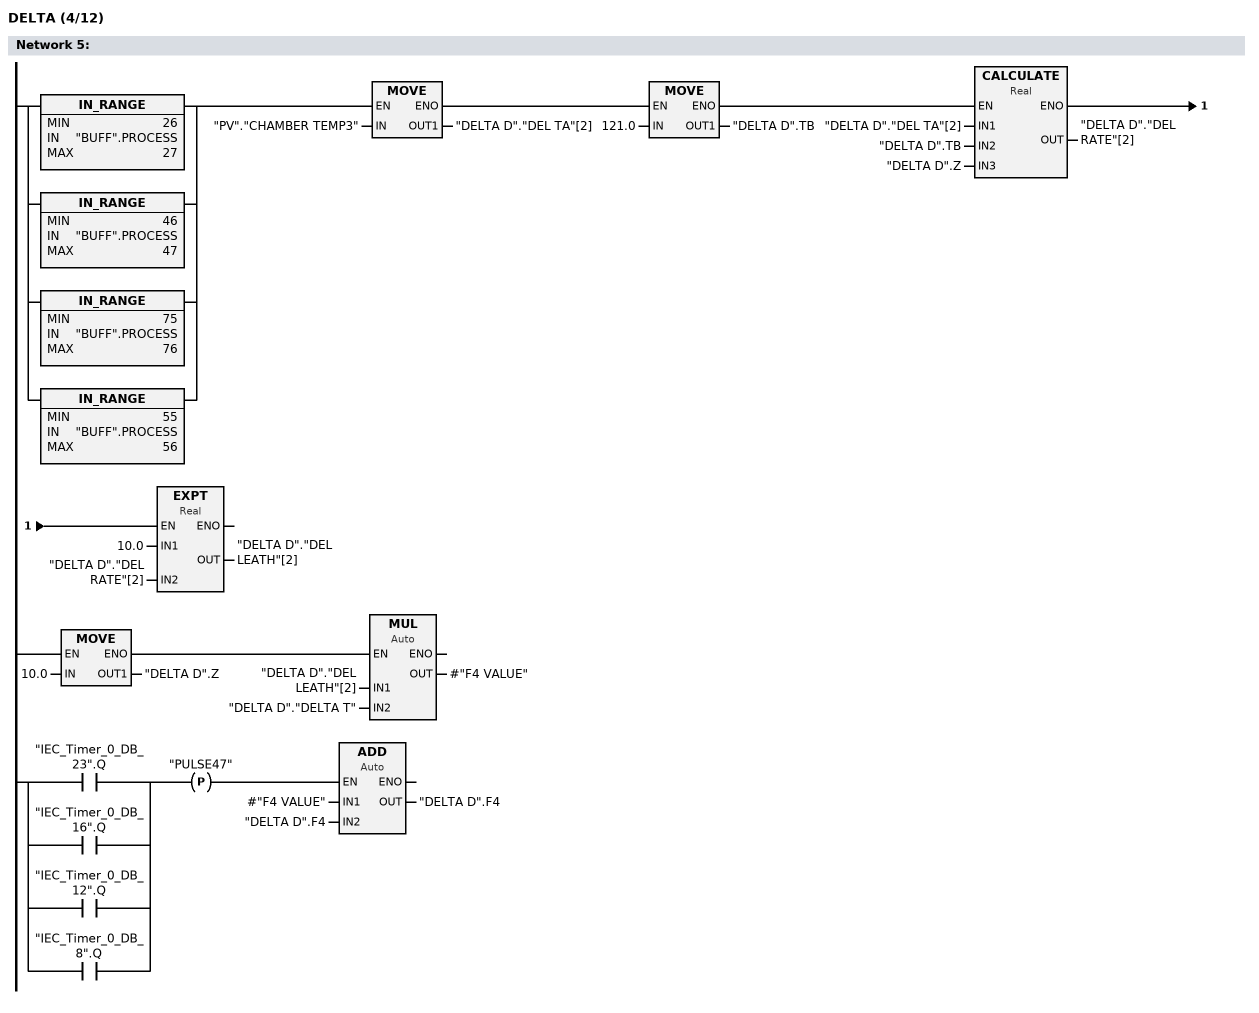
   IF ((26 <= "BUFF".PROCESS) AND ("BUFF".PROCESS <= 27)) OR ((46 <= "BUFF".PROCESS) AND ("BUFF".PROCESS <= 47)) OR ((75 <= "BUFF".PROCESS) AND ("BUFF".PROCESS <= 76)) OR ((55 <= "BUFF".PROCESS) AND ("BUFF".PROCESS <= 56)) THEN
       "DELTA D"."DEL TA"[2] := "PV"."CHAMBER TEMP3";
       "DELTA D".TB := 121.0;
       "DELTA D"."DEL RATE"[2] := ("DELTA D"."DEL TA"[2]-"DELTA D".TB)/"DELTA D".Z;
       "DELTA D"."DEL LEATH"[2] := 10.0 ** "DELTA D"."DEL RATE"[2];
   END_IF;
   "DELTA D".Z := 10.0;
   #"F4 VALUE" := "DELTA D"."DEL LEATH"[2] * "DELTA D"."DELTA T";
   #_w1 := "IEC_Timer_0_DB_23".Q OR "IEC_Timer_0_DB_16".Q OR "IEC_Timer_0_DB_12".Q OR "IEC_Timer_0_DB_8".Q;
   #_w2 := #_w1 AND NOT "PULSE47";   // rising edge
   "PULSE47" := #_w1;
   IF #_w2 THEN "DELTA D".F4 := #"F4 VALUE" + "DELTA D".F4; END_IF;
END_REGION

REGION Network 6
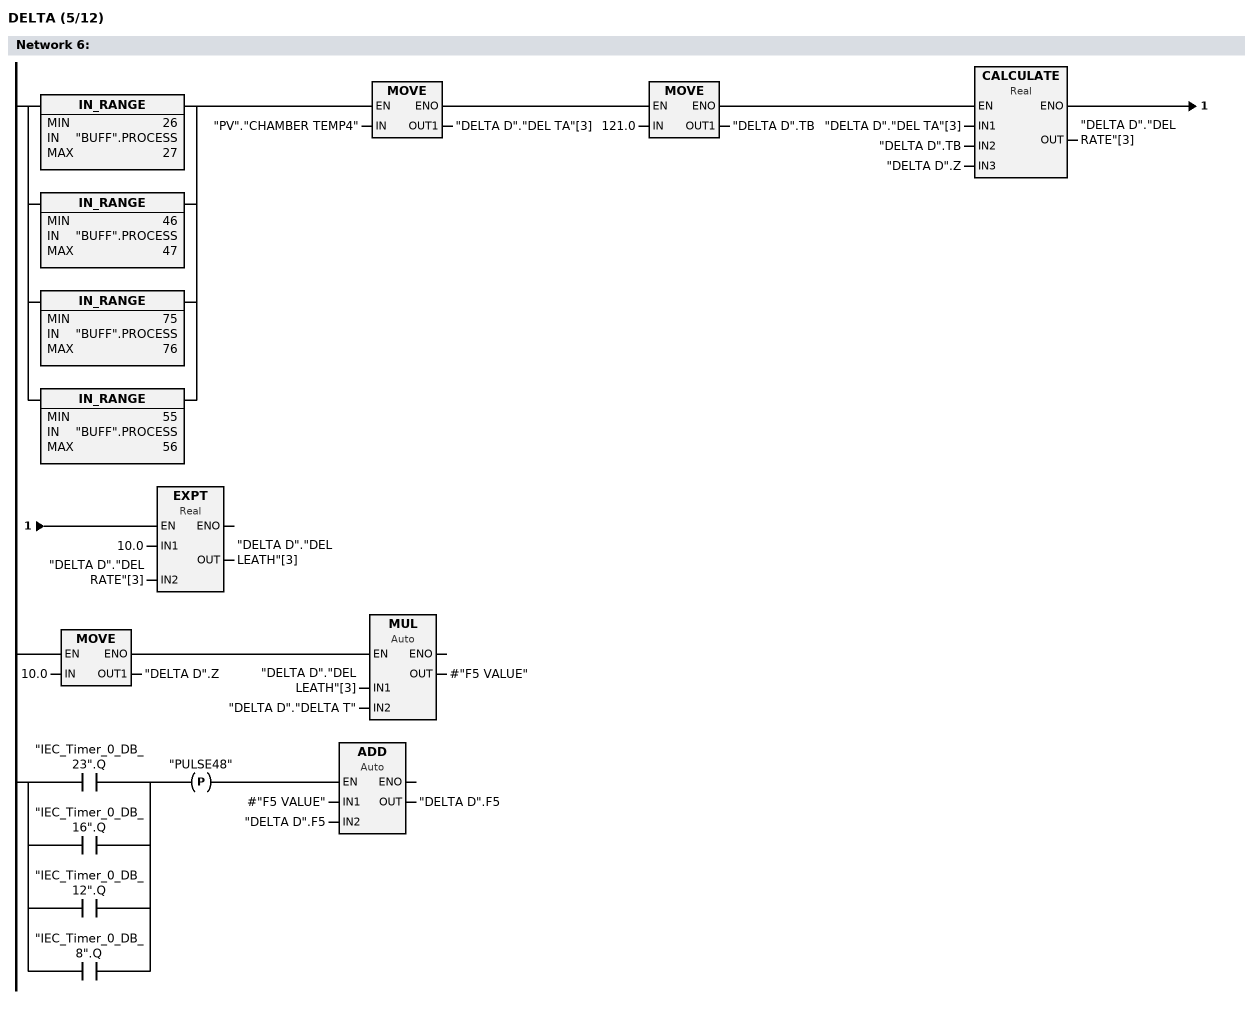
   IF ((26 <= "BUFF".PROCESS) AND ("BUFF".PROCESS <= 27)) OR ((46 <= "BUFF".PROCESS) AND ("BUFF".PROCESS <= 47)) OR ((75 <= "BUFF".PROCESS) AND ("BUFF".PROCESS <= 76)) OR ((55 <= "BUFF".PROCESS) AND ("BUFF".PROCESS <= 56)) THEN
       "DELTA D"."DEL TA"[3] := "PV"."CHAMBER TEMP4";
       "DELTA D".TB := 121.0;
       "DELTA D"."DEL RATE"[3] := ("DELTA D"."DEL TA"[3]-"DELTA D".TB)/"DELTA D".Z;
       "DELTA D"."DEL LEATH"[3] := 10.0 ** "DELTA D"."DEL RATE"[3];
   END_IF;
   "DELTA D".Z := 10.0;
   #"F5 VALUE" := "DELTA D"."DEL LEATH"[3] * "DELTA D"."DELTA T";
   #_w1 := "IEC_Timer_0_DB_23".Q OR "IEC_Timer_0_DB_16".Q OR "IEC_Timer_0_DB_12".Q OR "IEC_Timer_0_DB_8".Q;
   #_w2 := #_w1 AND NOT "PULSE48";   // rising edge
   "PULSE48" := #_w1;
   IF #_w2 THEN "DELTA D".F5 := #"F5 VALUE" + "DELTA D".F5; END_IF;
END_REGION

REGION Network 7
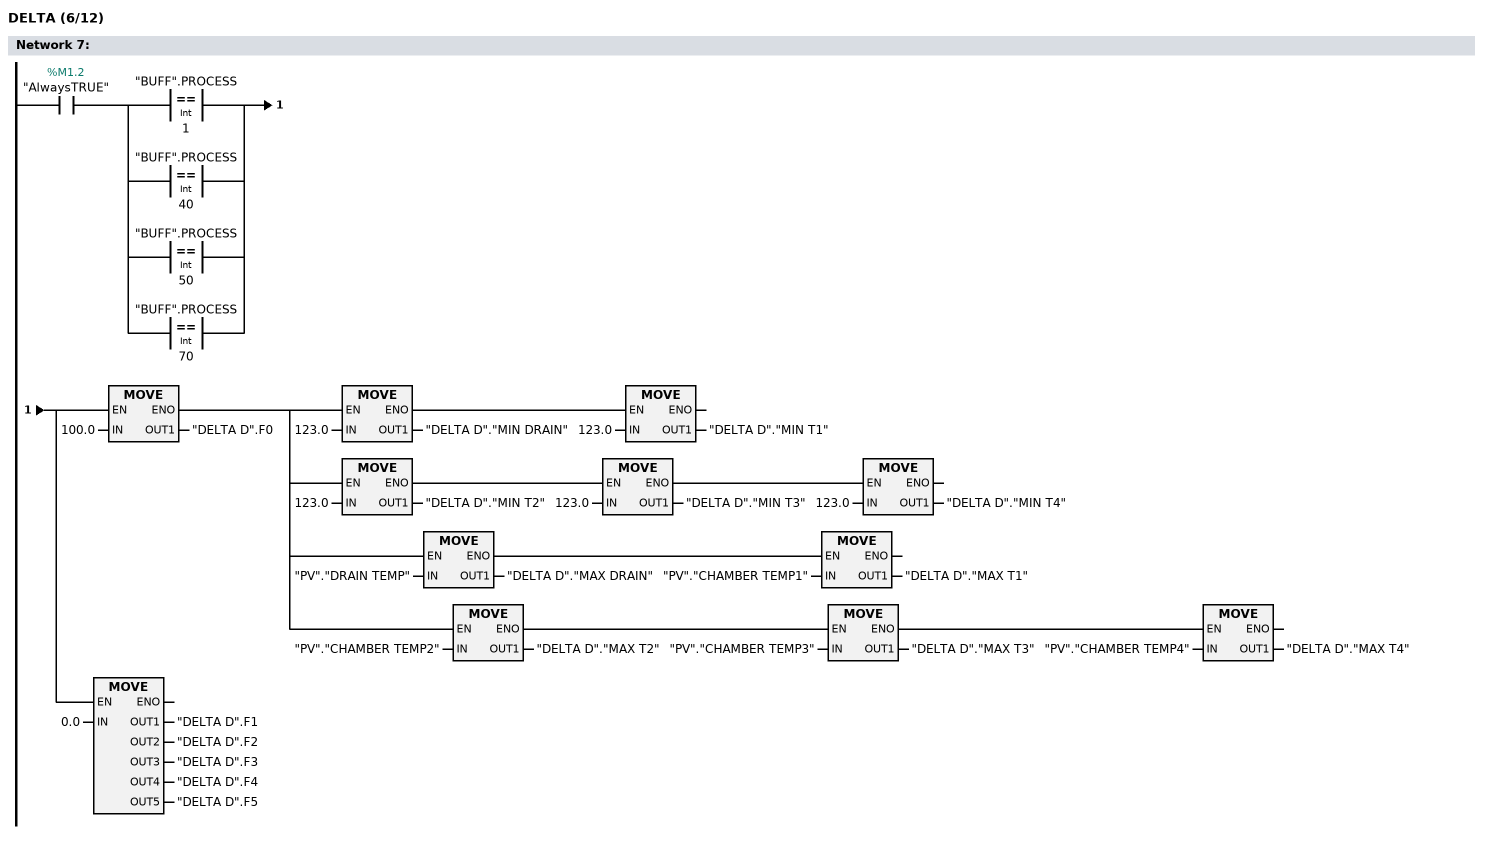
   RUNG wire#powerrail
      Contact( "AlwaysTRUE" )
      wire#w1
      { S7_Templates := "SrcType := Int" } EQ_Contact(in1 := "BUFF".PROCESS, in2 := 1)
      wire#w2
      Move(in := 100.0, out1 => "DELTA D".F0)
      wire#w3
      Move(in := 123.0, out1 => "DELTA D"."MIN DRAIN")
      Move(in := 123.0, out1 => "DELTA D"."MIN T1")
   END_RUNG
   RUNG wire#w1
      { S7_Templates := "SrcType := Int" } EQ_Contact(in1 := "BUFF".PROCESS, in2 := 40)
   END_RUNG wire#w2
   RUNG wire#w1
      { S7_Templates := "SrcType := Int" } EQ_Contact(in1 := "BUFF".PROCESS, in2 := 50)
   END_RUNG wire#w2
   RUNG wire#w1
      { S7_Templates := "SrcType := Int" } EQ_Contact(in1 := "BUFF".PROCESS, in2 := 70)
   END_RUNG wire#w2
   RUNG wire#w3
      Move(in := 123.0, out1 => "DELTA D"."MIN T2")
      Move(in := 123.0, out1 => "DELTA D"."MIN T3")
      Move(in := 123.0, out1 => "DELTA D"."MIN T4")
   END_RUNG
   RUNG wire#w3
      Move(in := "PV"."DRAIN TEMP", out1 => "DELTA D"."MAX DRAIN")
      Move(in := "PV"."CHAMBER TEMP1", out1 => "DELTA D"."MAX T1")
   END_RUNG
   RUNG wire#w3
      Move(in := "PV"."CHAMBER TEMP2", out1 => "DELTA D"."MAX T2")
      Move(in := "PV"."CHAMBER TEMP3", out1 => "DELTA D"."MAX T3")
      Move(in := "PV"."CHAMBER TEMP4", out1 => "DELTA D"."MAX T4")
   END_RUNG
   RUNG wire#w2
      Move(in := 0.0, out1 => "DELTA D".F1, out2 => "DELTA D".F2, out3 => "DELTA D".F3, out4 => "DELTA D".F4, out5 => "DELTA D".F5)
   END_RUNG
   // the same network as SCL:
   IF "AlwaysTRUE" AND (("BUFF".PROCESS = 1) OR ("BUFF".PROCESS = 40) OR ("BUFF".PROCESS = 50) OR ("BUFF".PROCESS = 70)) THEN
       "DELTA D".F0 := 100.0;
       "DELTA D"."MIN DRAIN" := 123.0;
       "DELTA D"."MIN T1" := 123.0;
       "DELTA D"."MIN T2" := 123.0;
       "DELTA D"."MIN T3" := 123.0;
       "DELTA D"."MIN T4" := 123.0;
       "DELTA D"."MAX DRAIN" := "PV"."DRAIN TEMP";
       "DELTA D"."MAX T1" := "PV"."CHAMBER TEMP1";
       "DELTA D"."MAX T2" := "PV"."CHAMBER TEMP2";
       "DELTA D"."MAX T3" := "PV"."CHAMBER TEMP3";
       "DELTA D"."MAX T4" := "PV"."CHAMBER TEMP4";
       "DELTA D".F1 := 0.0;
       "DELTA D".F2 := 0.0;
       "DELTA D".F3 := 0.0;
       "DELTA D".F4 := 0.0;
       "DELTA D".F5 := 0.0;
   END_IF;
END_REGION

REGION Network 8
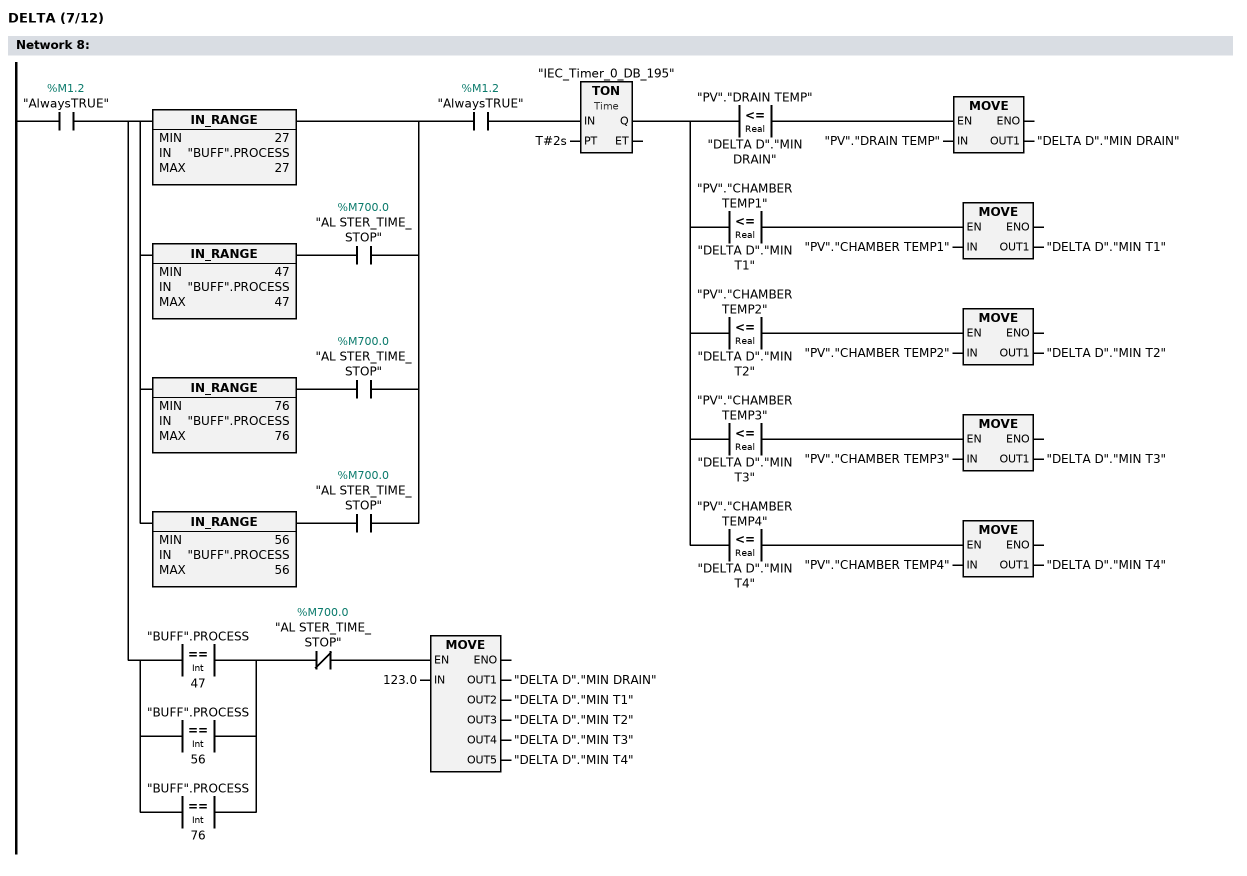
   RUNG wire#powerrail
      Contact( "AlwaysTRUE" )
      wire#w1
      { S7_Templates := "SrcType := Int" } InRange(min := 27, in := "BUFF".PROCESS, max := 27)
      wire#w2
      Contact( "AlwaysTRUE" )
      { S7_Templates := "time_type := Time" } "IEC_Timer_0_DB_195".TON(pt := T#2s, et =>)
      wire#w3
      { S7_Templates := "SrcType := Real" } LE_Contact(in1 := "PV"."DRAIN TEMP", in2 := "DELTA D"."MIN DRAIN")
      Move(in := "PV"."DRAIN TEMP", out1 => "DELTA D"."MIN DRAIN")
   END_RUNG
   RUNG wire#w1
      { S7_Templates := "SrcType := Int" } InRange(min := 47, in := "BUFF".PROCESS, max := 47)
      Contact( "AL STER_TIME_STOP" )
   END_RUNG wire#w2
   RUNG wire#w1
      { S7_Templates := "SrcType := Int" } InRange(min := 76, in := "BUFF".PROCESS, max := 76)
      Contact( "AL STER_TIME_STOP" )
   END_RUNG wire#w2
   RUNG wire#w1
      { S7_Templates := "SrcType := Int" } InRange(min := 56, in := "BUFF".PROCESS, max := 56)
      Contact( "AL STER_TIME_STOP" )
   END_RUNG wire#w2
   RUNG wire#w3
      { S7_Templates := "SrcType := Real" } LE_Contact(in1 := "PV"."CHAMBER TEMP1", in2 := "DELTA D"."MIN T1")
      Move(in := "PV"."CHAMBER TEMP1", out1 => "DELTA D"."MIN T1")
   END_RUNG
   RUNG wire#w3
      { S7_Templates := "SrcType := Real" } LE_Contact(in1 := "PV"."CHAMBER TEMP2", in2 := "DELTA D"."MIN T2")
      Move(in := "PV"."CHAMBER TEMP2", out1 => "DELTA D"."MIN T2")
   END_RUNG
   RUNG wire#w3
      { S7_Templates := "SrcType := Real" } LE_Contact(in1 := "PV"."CHAMBER TEMP3", in2 := "DELTA D"."MIN T3")
      Move(in := "PV"."CHAMBER TEMP3", out1 => "DELTA D"."MIN T3")
   END_RUNG
   RUNG wire#w3
      { S7_Templates := "SrcType := Real" } LE_Contact(in1 := "PV"."CHAMBER TEMP4", in2 := "DELTA D"."MIN T4")
      Move(in := "PV"."CHAMBER TEMP4", out1 => "DELTA D"."MIN T4")
   END_RUNG
   RUNG wire#w1
      { S7_Templates := "SrcType := Int" } EQ_Contact(in1 := "BUFF".PROCESS, in2 := 47)
      wire#w4
      I_Contact( "AL STER_TIME_STOP" )
      Move(in := 123.0, out1 => "DELTA D"."MIN DRAIN", out2 => "DELTA D"."MIN T1", out3 => "DELTA D"."MIN T2", out4 => "DELTA D"."MIN T3", out5 => "DELTA D"."MIN T4")
   END_RUNG
   RUNG wire#w1
      { S7_Templates := "SrcType := Int" } EQ_Contact(in1 := "BUFF".PROCESS, in2 := 56)
   END_RUNG wire#w4
   RUNG wire#w1
      { S7_Templates := "SrcType := Int" } EQ_Contact(in1 := "BUFF".PROCESS, in2 := 76)
   END_RUNG wire#w4
   // the same network as SCL:
   "IEC_Timer_0_DB_195".TON(IN := "AlwaysTRUE" AND (((27 <= "BUFF".PROCESS) AND ("BUFF".PROCESS <= 27)) OR ((47 <= "BUFF".PROCESS) AND ("BUFF".PROCESS <= 47) AND "AL STER_TIME_STOP") OR ((76 <= "BUFF".PROCESS) AND ("BUFF".PROCESS <= 76) AND "AL STER_TIME_STOP") OR ((56 <= "BUFF".PROCESS) AND ("BUFF".PROCESS <= 56) AND "AL STER_TIME_STOP")) AND "AlwaysTRUE",
                           PT := T#2s);
   IF "IEC_Timer_0_DB_195".Q AND ("PV"."DRAIN TEMP" <= "DELTA D"."MIN DRAIN") THEN
       "DELTA D"."MIN DRAIN" := "PV"."DRAIN TEMP";
   END_IF;
   IF "IEC_Timer_0_DB_195".Q AND ("PV"."CHAMBER TEMP1" <= "DELTA D"."MIN T1") THEN
       "DELTA D"."MIN T1" := "PV"."CHAMBER TEMP1";
   END_IF;
   IF "IEC_Timer_0_DB_195".Q AND ("PV"."CHAMBER TEMP2" <= "DELTA D"."MIN T2") THEN
       "DELTA D"."MIN T2" := "PV"."CHAMBER TEMP2";
   END_IF;
   IF "IEC_Timer_0_DB_195".Q AND ("PV"."CHAMBER TEMP3" <= "DELTA D"."MIN T3") THEN
       "DELTA D"."MIN T3" := "PV"."CHAMBER TEMP3";
   END_IF;
   IF "IEC_Timer_0_DB_195".Q AND ("PV"."CHAMBER TEMP4" <= "DELTA D"."MIN T4") THEN
       "DELTA D"."MIN T4" := "PV"."CHAMBER TEMP4";
   END_IF;
   IF "AlwaysTRUE" AND (("BUFF".PROCESS = 47) OR ("BUFF".PROCESS = 56) OR ("BUFF".PROCESS = 76)) AND NOT "AL STER_TIME_STOP" THEN
       "DELTA D"."MIN DRAIN" := 123.0;
       "DELTA D"."MIN T1" := 123.0;
       "DELTA D"."MIN T2" := 123.0;
       "DELTA D"."MIN T3" := 123.0;
       "DELTA D"."MIN T4" := 123.0;
   END_IF;
END_REGION

REGION Network 9
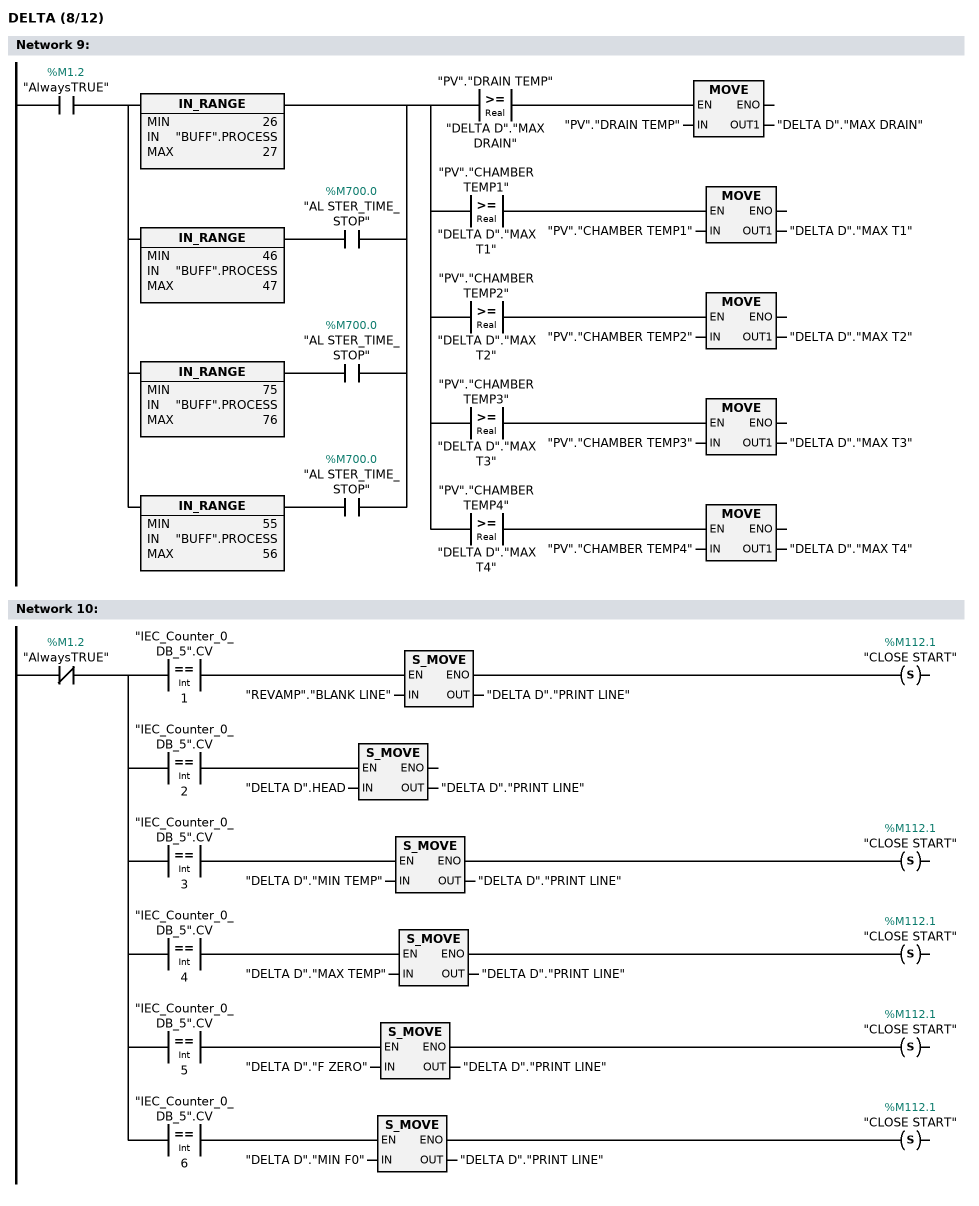
   RUNG wire#powerrail
      Contact( "AlwaysTRUE" )
      wire#w1
      { S7_Templates := "SrcType := Int" } InRange(min := 26, in := "BUFF".PROCESS, max := 27)
      wire#w2
      { S7_Templates := "SrcType := Real" } GE_Contact(in1 := "PV"."DRAIN TEMP", in2 := "DELTA D"."MAX DRAIN")
      Move(in := "PV"."DRAIN TEMP", out1 => "DELTA D"."MAX DRAIN")
   END_RUNG
   RUNG wire#w1
      { S7_Templates := "SrcType := Int" } InRange(min := 46, in := "BUFF".PROCESS, max := 47)
      Contact( "AL STER_TIME_STOP" )
   END_RUNG wire#w2
   RUNG wire#w1
      { S7_Templates := "SrcType := Int" } InRange(min := 75, in := "BUFF".PROCESS, max := 76)
      Contact( "AL STER_TIME_STOP" )
   END_RUNG wire#w2
   RUNG wire#w1
      { S7_Templates := "SrcType := Int" } InRange(min := 55, in := "BUFF".PROCESS, max := 56)
      Contact( "AL STER_TIME_STOP" )
   END_RUNG wire#w2
   RUNG wire#w2
      { S7_Templates := "SrcType := Real" } GE_Contact(in1 := "PV"."CHAMBER TEMP1", in2 := "DELTA D"."MAX T1")
      Move(in := "PV"."CHAMBER TEMP1", out1 => "DELTA D"."MAX T1")
   END_RUNG
   RUNG wire#w2
      { S7_Templates := "SrcType := Real" } GE_Contact(in1 := "PV"."CHAMBER TEMP2", in2 := "DELTA D"."MAX T2")
      Move(in := "PV"."CHAMBER TEMP2", out1 => "DELTA D"."MAX T2")
   END_RUNG
   RUNG wire#w2
      { S7_Templates := "SrcType := Real" } GE_Contact(in1 := "PV"."CHAMBER TEMP3", in2 := "DELTA D"."MAX T3")
      Move(in := "PV"."CHAMBER TEMP3", out1 => "DELTA D"."MAX T3")
   END_RUNG
   RUNG wire#w2
      { S7_Templates := "SrcType := Real" } GE_Contact(in1 := "PV"."CHAMBER TEMP4", in2 := "DELTA D"."MAX T4")
      Move(in := "PV"."CHAMBER TEMP4", out1 => "DELTA D"."MAX T4")
   END_RUNG
   // the same network as SCL:
   #_w1 := "AlwaysTRUE" AND (((26 <= "BUFF".PROCESS) AND ("BUFF".PROCESS <= 27)) OR ((46 <= "BUFF".PROCESS) AND ("BUFF".PROCESS <= 47) AND "AL STER_TIME_STOP") OR ((75 <= "BUFF".PROCESS) AND ("BUFF".PROCESS <= 76) AND "AL STER_TIME_STOP") OR ((55 <= "BUFF".PROCESS) AND ("BUFF".PROCESS <= 56) AND "AL STER_TIME_STOP"));
   IF #_w1 AND ("PV"."DRAIN TEMP" >= "DELTA D"."MAX DRAIN") THEN
       "DELTA D"."MAX DRAIN" := "PV"."DRAIN TEMP";
   END_IF;
   IF #_w1 AND ("PV"."CHAMBER TEMP1" >= "DELTA D"."MAX T1") THEN
       "DELTA D"."MAX T1" := "PV"."CHAMBER TEMP1";
   END_IF;
   IF #_w1 AND ("PV"."CHAMBER TEMP2" >= "DELTA D"."MAX T2") THEN
       "DELTA D"."MAX T2" := "PV"."CHAMBER TEMP2";
   END_IF;
   IF #_w1 AND ("PV"."CHAMBER TEMP3" >= "DELTA D"."MAX T3") THEN
       "DELTA D"."MAX T3" := "PV"."CHAMBER TEMP3";
   END_IF;
   IF #_w1 AND ("PV"."CHAMBER TEMP4" >= "DELTA D"."MAX T4") THEN
       "DELTA D"."MAX T4" := "PV"."CHAMBER TEMP4";
   END_IF;
END_REGION

REGION Network 10
   RUNG wire#powerrail
      I_Contact( "AlwaysTRUE" )
      wire#w1
      { S7_Templates := "SrcType := Int" } EQ_Contact(in1 := "IEC_Counter_0_DB_5".CV, in2 := 1)
      S_Move(in := "REVAMP"."BLANK LINE", out => "DELTA D"."PRINT LINE")
      S_Coil( "CLOSE START" )
   END_RUNG
   RUNG wire#w1
      { S7_Templates := "SrcType := Int" } EQ_Contact(in1 := "IEC_Counter_0_DB_5".CV, in2 := 2)
      S_Move(in := "DELTA D".HEAD, out => "DELTA D"."PRINT LINE")
   END_RUNG
   RUNG wire#w1
      { S7_Templates := "SrcType := Int" } EQ_Contact(in1 := "IEC_Counter_0_DB_5".CV, in2 := 3)
      S_Move(in := "DELTA D"."MIN TEMP", out => "DELTA D"."PRINT LINE")
      S_Coil( "CLOSE START" )
   END_RUNG
   RUNG wire#w1
      { S7_Templates := "SrcType := Int" } EQ_Contact(in1 := "IEC_Counter_0_DB_5".CV, in2 := 4)
      S_Move(in := "DELTA D"."MAX TEMP", out => "DELTA D"."PRINT LINE")
      S_Coil( "CLOSE START" )
   END_RUNG
   RUNG wire#w1
      { S7_Templates := "SrcType := Int" } EQ_Contact(in1 := "IEC_Counter_0_DB_5".CV, in2 := 5)
      S_Move(in := "DELTA D"."F ZERO", out => "DELTA D"."PRINT LINE")
      S_Coil( "CLOSE START" )
   END_RUNG
   RUNG wire#w1
      { S7_Templates := "SrcType := Int" } EQ_Contact(in1 := "IEC_Counter_0_DB_5".CV, in2 := 6)
      S_Move(in := "DELTA D"."MIN F0", out => "DELTA D"."PRINT LINE")
      S_Coil( "CLOSE START" )
   END_RUNG
   // the same network as SCL:
   IF NOT "AlwaysTRUE" AND ("IEC_Counter_0_DB_5".CV = 1) THEN
       "DELTA D"."PRINT LINE" := "REVAMP"."BLANK LINE";
       "CLOSE START" := TRUE;
   END_IF;
   IF NOT "AlwaysTRUE" AND ("IEC_Counter_0_DB_5".CV = 2) THEN
       "DELTA D"."PRINT LINE" := "DELTA D".HEAD;
   END_IF;
   IF NOT "AlwaysTRUE" AND ("IEC_Counter_0_DB_5".CV = 3) THEN
       "DELTA D"."PRINT LINE" := "DELTA D"."MIN TEMP";
       "CLOSE START" := TRUE;
   END_IF;
   IF NOT "AlwaysTRUE" AND ("IEC_Counter_0_DB_5".CV = 4) THEN
       "DELTA D"."PRINT LINE" := "DELTA D"."MAX TEMP";
       "CLOSE START" := TRUE;
   END_IF;
   IF NOT "AlwaysTRUE" AND ("IEC_Counter_0_DB_5".CV = 5) THEN
       "DELTA D"."PRINT LINE" := "DELTA D"."F ZERO";
       "CLOSE START" := TRUE;
   END_IF;
   IF NOT "AlwaysTRUE" AND ("IEC_Counter_0_DB_5".CV = 6) THEN
       "DELTA D"."PRINT LINE" := "DELTA D"."MIN F0";
       "CLOSE START" := TRUE;
   END_IF;
END_REGION

REGION Network 11
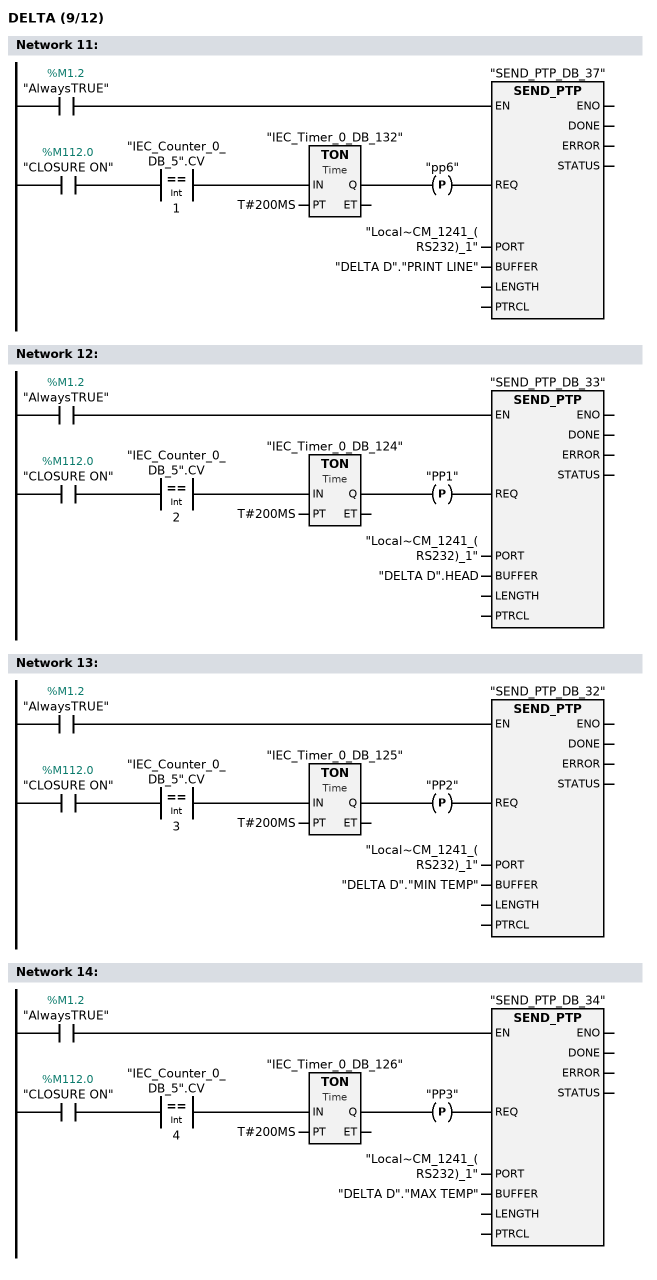
   RUNG wire#powerrail
      Contact( "AlwaysTRUE" )
      "SEND_PTP_DB_37".SEND_PTP(REQ := wire#w1, PORT := "Local~CM_1241_(RS232)_1", BUFFER := "DELTA D"."PRINT LINE", LENGTH :=, PTRCL :=, DONE =>, ERROR =>, STATUS =>)
   END_RUNG
   RUNG wire#powerrail
      Contact( "CLOSURE ON" )
      { S7_Templates := "SrcType := Int" } EQ_Contact(in1 := "IEC_Counter_0_DB_5".CV, in2 := 1)
      { S7_Templates := "time_type := Time" } "IEC_Timer_0_DB_132".TON(pt := T#200MS, et =>)
      P_Trig( "pp6" )
   END_RUNG wire#w1
   // the same network as SCL:
   "IEC_Timer_0_DB_132".TON(IN := "CLOSURE ON" AND ("IEC_Counter_0_DB_5".CV = 1), PT := T#200MS);
   #_w1 := "IEC_Timer_0_DB_132".Q AND NOT "pp6";   // rising edge
   "pp6" := "IEC_Timer_0_DB_132".Q;
   IF "AlwaysTRUE" THEN
       "SEND_PTP_DB_37"(REQ := #_w1, PORT := "Local~CM_1241_(RS232)_1", BUFFER := "DELTA D"."PRINT LINE");   // SEND_PTP
   END_IF;
END_REGION

REGION Network 12
   RUNG wire#powerrail
      Contact( "AlwaysTRUE" )
      "SEND_PTP_DB_33".SEND_PTP(REQ := wire#w1, PORT := "Local~CM_1241_(RS232)_1", BUFFER := "DELTA D".HEAD, LENGTH :=, PTRCL :=, DONE =>, ERROR =>, STATUS =>)
   END_RUNG
   RUNG wire#powerrail
      Contact( "CLOSURE ON" )
      { S7_Templates := "SrcType := Int" } EQ_Contact(in1 := "IEC_Counter_0_DB_5".CV, in2 := 2)
      { S7_Templates := "time_type := Time" } "IEC_Timer_0_DB_124".TON(pt := T#200MS, et =>)
      P_Trig( "PP1" )
   END_RUNG wire#w1
   // the same network as SCL:
   "IEC_Timer_0_DB_124".TON(IN := "CLOSURE ON" AND ("IEC_Counter_0_DB_5".CV = 2), PT := T#200MS);
   #_w1 := "IEC_Timer_0_DB_124".Q AND NOT "PP1";   // rising edge
   "PP1" := "IEC_Timer_0_DB_124".Q;
   IF "AlwaysTRUE" THEN
       "SEND_PTP_DB_33"(REQ := #_w1, PORT := "Local~CM_1241_(RS232)_1", BUFFER := "DELTA D".HEAD);   // SEND_PTP
   END_IF;
END_REGION

REGION Network 13
   RUNG wire#powerrail
      Contact( "AlwaysTRUE" )
      "SEND_PTP_DB_32".SEND_PTP(REQ := wire#w1, PORT := "Local~CM_1241_(RS232)_1", BUFFER := "DELTA D"."MIN TEMP", LENGTH :=, PTRCL :=, DONE =>, ERROR =>, STATUS =>)
   END_RUNG
   RUNG wire#powerrail
      Contact( "CLOSURE ON" )
      { S7_Templates := "SrcType := Int" } EQ_Contact(in1 := "IEC_Counter_0_DB_5".CV, in2 := 3)
      { S7_Templates := "time_type := Time" } "IEC_Timer_0_DB_125".TON(pt := T#200MS, et =>)
      P_Trig( "PP2" )
   END_RUNG wire#w1
   // the same network as SCL:
   "IEC_Timer_0_DB_125".TON(IN := "CLOSURE ON" AND ("IEC_Counter_0_DB_5".CV = 3), PT := T#200MS);
   #_w1 := "IEC_Timer_0_DB_125".Q AND NOT "PP2";   // rising edge
   "PP2" := "IEC_Timer_0_DB_125".Q;
   IF "AlwaysTRUE" THEN
       "SEND_PTP_DB_32"(REQ := #_w1, PORT := "Local~CM_1241_(RS232)_1", BUFFER := "DELTA D"."MIN TEMP");   // SEND_PTP
   END_IF;
END_REGION

REGION Network 14
   RUNG wire#powerrail
      Contact( "AlwaysTRUE" )
      "SEND_PTP_DB_34".SEND_PTP(REQ := wire#w1, PORT := "Local~CM_1241_(RS232)_1", BUFFER := "DELTA D"."MAX TEMP", LENGTH :=, PTRCL :=, DONE =>, ERROR =>, STATUS =>)
   END_RUNG
   RUNG wire#powerrail
      Contact( "CLOSURE ON" )
      { S7_Templates := "SrcType := Int" } EQ_Contact(in1 := "IEC_Counter_0_DB_5".CV, in2 := 4)
      { S7_Templates := "time_type := Time" } "IEC_Timer_0_DB_126".TON(pt := T#200MS, et =>)
      P_Trig( "PP3" )
   END_RUNG wire#w1
   // the same network as SCL:
   "IEC_Timer_0_DB_126".TON(IN := "CLOSURE ON" AND ("IEC_Counter_0_DB_5".CV = 4), PT := T#200MS);
   #_w1 := "IEC_Timer_0_DB_126".Q AND NOT "PP3";   // rising edge
   "PP3" := "IEC_Timer_0_DB_126".Q;
   IF "AlwaysTRUE" THEN
       "SEND_PTP_DB_34"(REQ := #_w1, PORT := "Local~CM_1241_(RS232)_1", BUFFER := "DELTA D"."MAX TEMP");   // SEND_PTP
   END_IF;
END_REGION

REGION Network 15
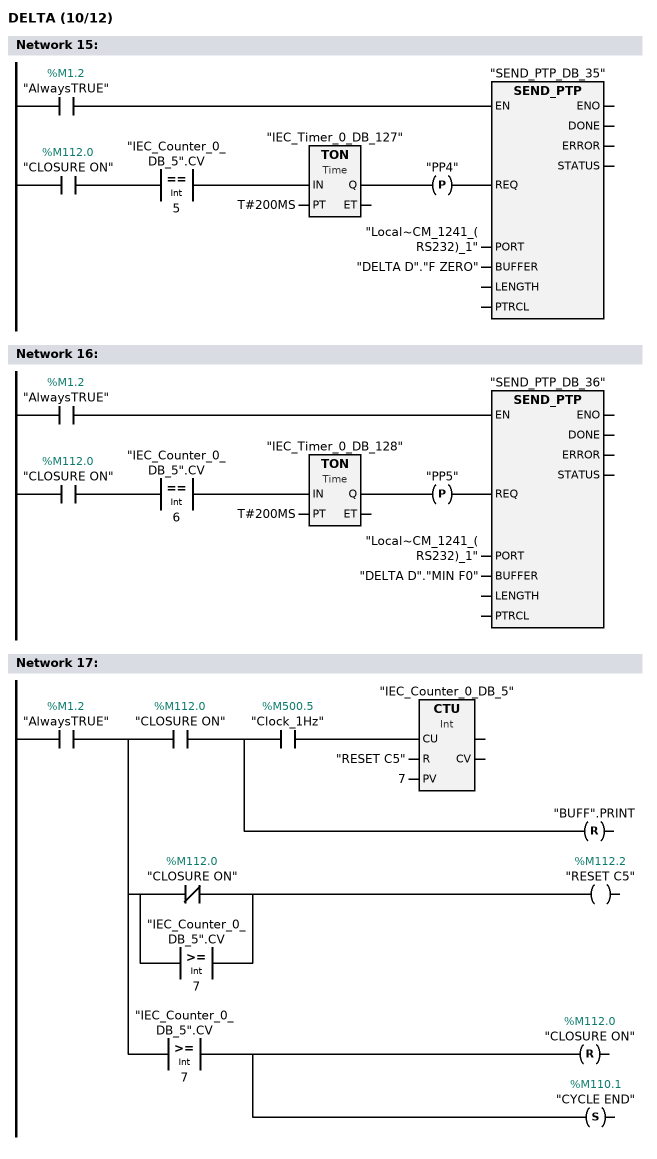
   RUNG wire#powerrail
      Contact( "AlwaysTRUE" )
      "SEND_PTP_DB_35".SEND_PTP(REQ := wire#w1, PORT := "Local~CM_1241_(RS232)_1", BUFFER := "DELTA D"."F ZERO", LENGTH :=, PTRCL :=, DONE =>, ERROR =>, STATUS =>)
   END_RUNG
   RUNG wire#powerrail
      Contact( "CLOSURE ON" )
      { S7_Templates := "SrcType := Int" } EQ_Contact(in1 := "IEC_Counter_0_DB_5".CV, in2 := 5)
      { S7_Templates := "time_type := Time" } "IEC_Timer_0_DB_127".TON(pt := T#200MS, et =>)
      P_Trig( "PP4" )
   END_RUNG wire#w1
   // the same network as SCL:
   "IEC_Timer_0_DB_127".TON(IN := "CLOSURE ON" AND ("IEC_Counter_0_DB_5".CV = 5), PT := T#200MS);
   #_w1 := "IEC_Timer_0_DB_127".Q AND NOT "PP4";   // rising edge
   "PP4" := "IEC_Timer_0_DB_127".Q;
   IF "AlwaysTRUE" THEN
       "SEND_PTP_DB_35"(REQ := #_w1, PORT := "Local~CM_1241_(RS232)_1", BUFFER := "DELTA D"."F ZERO");   // SEND_PTP
   END_IF;
END_REGION

REGION Network 16
   RUNG wire#powerrail
      Contact( "AlwaysTRUE" )
      "SEND_PTP_DB_36".SEND_PTP(REQ := wire#w1, PORT := "Local~CM_1241_(RS232)_1", BUFFER := "DELTA D"."MIN F0", LENGTH :=, PTRCL :=, DONE =>, ERROR =>, STATUS =>)
   END_RUNG
   RUNG wire#powerrail
      Contact( "CLOSURE ON" )
      { S7_Templates := "SrcType := Int" } EQ_Contact(in1 := "IEC_Counter_0_DB_5".CV, in2 := 6)
      { S7_Templates := "time_type := Time" } "IEC_Timer_0_DB_128".TON(pt := T#200MS, et =>)
      P_Trig( "PP5" )
   END_RUNG wire#w1
   // the same network as SCL:
   "IEC_Timer_0_DB_128".TON(IN := "CLOSURE ON" AND ("IEC_Counter_0_DB_5".CV = 6), PT := T#200MS);
   #_w1 := "IEC_Timer_0_DB_128".Q AND NOT "PP5";   // rising edge
   "PP5" := "IEC_Timer_0_DB_128".Q;
   IF "AlwaysTRUE" THEN
       "SEND_PTP_DB_36"(REQ := #_w1, PORT := "Local~CM_1241_(RS232)_1", BUFFER := "DELTA D"."MIN F0");   // SEND_PTP
   END_IF;
END_REGION

REGION Network 17
   RUNG wire#powerrail
      Contact( "AlwaysTRUE" )
      wire#w1
      Contact( "CLOSURE ON" )
      wire#w2
      Contact( "Clock_1Hz" )
      { S7_Templates := "value_type := Int" } "IEC_Counter_0_DB_5".CTU(r := "RESET C5", pv := 7, cv =>)
   END_RUNG
   RUNG wire#w2
      R_Coil( "BUFF".PRINT )
   END_RUNG
   RUNG wire#w1
      I_Contact( "CLOSURE ON" )
      wire#w3
      Coil( "RESET C5" )
   END_RUNG
   RUNG wire#w1
      { S7_Templates := "SrcType := Int" } GE_Contact(in1 := "IEC_Counter_0_DB_5".CV, in2 := 7)
   END_RUNG wire#w3
   RUNG wire#w1
      { S7_Templates := "SrcType := Int" } GE_Contact(in1 := "IEC_Counter_0_DB_5".CV, in2 := 7)
      wire#w4
      R_Coil( "CLOSURE ON" )
   END_RUNG
   RUNG wire#w4
      S_Coil( "CYCLE END" )
   END_RUNG
   // the same network as SCL:
   #_w1 := "AlwaysTRUE" AND "CLOSURE ON";
   "IEC_Counter_0_DB_5".CTU(CU := #_w1 AND "Clock_1Hz", R := "RESET C5", PV := 7);
   IF #_w1 THEN "BUFF".PRINT := FALSE; END_IF;
   "RESET C5" := "AlwaysTRUE" AND (NOT "CLOSURE ON" OR ("IEC_Counter_0_DB_5".CV >= 7));
   IF "AlwaysTRUE" AND ("IEC_Counter_0_DB_5".CV >= 7) THEN
       "CLOSURE ON" := FALSE;
       "CYCLE END" := TRUE;
   END_IF;
END_REGION

REGION Network 18
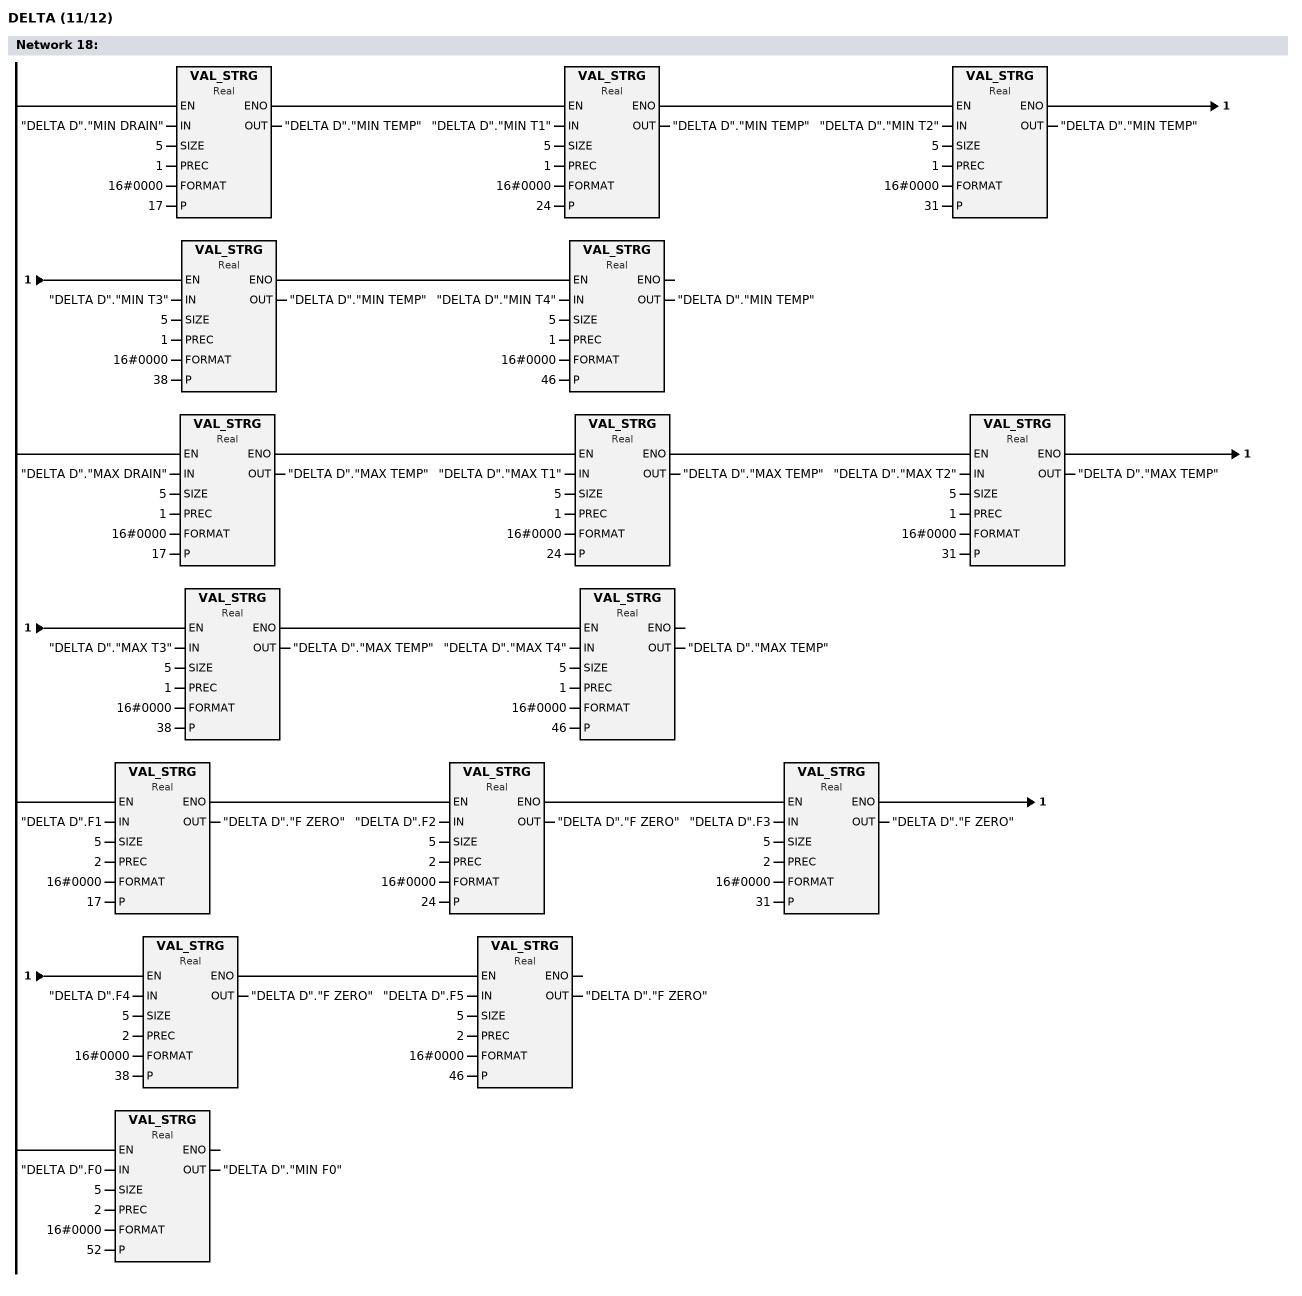
   RUNG wire#powerrail
      { S7_Templates := "[value_type := Real, str_type := String]" } VAL_STRG(IN := "DELTA D"."MIN DRAIN", SIZE := 5, PREC := 1, FORMAT := 16#0000, P := 17, OUT => "DELTA D"."MIN TEMP")
      { S7_Templates := "[value_type := Real, str_type := String]" } VAL_STRG(IN := "DELTA D"."MIN T1", SIZE := 5, PREC := 1, FORMAT := 16#0000, P := 24, OUT => "DELTA D"."MIN TEMP")
      { S7_Templates := "[value_type := Real, str_type := String]" } VAL_STRG(IN := "DELTA D"."MIN T2", SIZE := 5, PREC := 1, FORMAT := 16#0000, P := 31, OUT => "DELTA D"."MIN TEMP")
      { S7_Templates := "[value_type := Real, str_type := String]" } VAL_STRG(IN := "DELTA D"."MIN T3", SIZE := 5, PREC := 1, FORMAT := 16#0000, P := 38, OUT => "DELTA D"."MIN TEMP")
      { S7_Templates := "[value_type := Real, str_type := String]" } VAL_STRG(IN := "DELTA D"."MIN T4", SIZE := 5, PREC := 1, FORMAT := 16#0000, P := 46, OUT => "DELTA D"."MIN TEMP")
   END_RUNG
   RUNG wire#powerrail
      { S7_Templates := "[value_type := Real, str_type := String]" } VAL_STRG(IN := "DELTA D"."MAX DRAIN", SIZE := 5, PREC := 1, FORMAT := 16#0000, P := 17, OUT => "DELTA D"."MAX TEMP")
      { S7_Templates := "[value_type := Real, str_type := String]" } VAL_STRG(IN := "DELTA D"."MAX T1", SIZE := 5, PREC := 1, FORMAT := 16#0000, P := 24, OUT => "DELTA D"."MAX TEMP")
      { S7_Templates := "[value_type := Real, str_type := String]" } VAL_STRG(IN := "DELTA D"."MAX T2", SIZE := 5, PREC := 1, FORMAT := 16#0000, P := 31, OUT => "DELTA D"."MAX TEMP")
      { S7_Templates := "[value_type := Real, str_type := String]" } VAL_STRG(IN := "DELTA D"."MAX T3", SIZE := 5, PREC := 1, FORMAT := 16#0000, P := 38, OUT => "DELTA D"."MAX TEMP")
      { S7_Templates := "[value_type := Real, str_type := String]" } VAL_STRG(IN := "DELTA D"."MAX T4", SIZE := 5, PREC := 1, FORMAT := 16#0000, P := 46, OUT => "DELTA D"."MAX TEMP")
   END_RUNG
   RUNG wire#powerrail
      { S7_Templates := "[value_type := Real, str_type := String]" } VAL_STRG(IN := "DELTA D".F1, SIZE := 5, PREC := 2, FORMAT := 16#0000, P := 17, OUT => "DELTA D"."F ZERO")
      { S7_Templates := "[value_type := Real, str_type := String]" } VAL_STRG(IN := "DELTA D".F2, SIZE := 5, PREC := 2, FORMAT := 16#0000, P := 24, OUT => "DELTA D"."F ZERO")
      { S7_Templates := "[value_type := Real, str_type := String]" } VAL_STRG(IN := "DELTA D".F3, SIZE := 5, PREC := 2, FORMAT := 16#0000, P := 31, OUT => "DELTA D"."F ZERO")
      { S7_Templates := "[value_type := Real, str_type := String]" } VAL_STRG(IN := "DELTA D".F4, SIZE := 5, PREC := 2, FORMAT := 16#0000, P := 38, OUT => "DELTA D"."F ZERO")
      { S7_Templates := "[value_type := Real, str_type := String]" } VAL_STRG(IN := "DELTA D".F5, SIZE := 5, PREC := 2, FORMAT := 16#0000, P := 46, OUT => "DELTA D"."F ZERO")
   END_RUNG
   RUNG wire#powerrail
      { S7_Templates := "[value_type := Real, str_type := String]" } VAL_STRG(IN := "DELTA D".F0, SIZE := 5, PREC := 2, FORMAT := 16#0000, P := 52, OUT => "DELTA D"."MIN F0")
   END_RUNG
   // the same network as SCL:
   VAL_STRG(IN := "DELTA D"."MIN DRAIN",
            SIZE := 5,
            PREC := 1,
            FORMAT := 16#0000,
            P := 17,
            OUT => "DELTA D"."MIN TEMP",
            ENO => #_w1);
   VAL_STRG(EN := #_w1,
            IN := "DELTA D"."MIN T1",
            SIZE := 5,
            PREC := 1,
            FORMAT := 16#0000,
            P := 24,
            OUT => "DELTA D"."MIN TEMP",
            ENO => #_w2);
   VAL_STRG(EN := #_w2,
            IN := "DELTA D"."MIN T2",
            SIZE := 5,
            PREC := 1,
            FORMAT := 16#0000,
            P := 31,
            OUT => "DELTA D"."MIN TEMP",
            ENO => #_w3);
   VAL_STRG(EN := #_w3,
            IN := "DELTA D"."MIN T3",
            SIZE := 5,
            PREC := 1,
            FORMAT := 16#0000,
            P := 38,
            OUT => "DELTA D"."MIN TEMP",
            ENO => #_w4);
   IF #_w4 THEN
       VAL_STRG(IN := "DELTA D"."MIN T4",
                SIZE := 5,
                PREC := 1,
                FORMAT := 16#0000,
                P := 46,
                OUT => "DELTA D"."MIN TEMP");
   END_IF;
   VAL_STRG(IN := "DELTA D"."MAX DRAIN",
            SIZE := 5,
            PREC := 1,
            FORMAT := 16#0000,
            P := 17,
            OUT => "DELTA D"."MAX TEMP",
            ENO => #_w5);
   VAL_STRG(EN := #_w5,
            IN := "DELTA D"."MAX T1",
            SIZE := 5,
            PREC := 1,
            FORMAT := 16#0000,
            P := 24,
            OUT => "DELTA D"."MAX TEMP",
            ENO => #_w6);
   VAL_STRG(EN := #_w6,
            IN := "DELTA D"."MAX T2",
            SIZE := 5,
            PREC := 1,
            FORMAT := 16#0000,
            P := 31,
            OUT => "DELTA D"."MAX TEMP",
            ENO => #_w7);
   VAL_STRG(EN := #_w7,
            IN := "DELTA D"."MAX T3",
            SIZE := 5,
            PREC := 1,
            FORMAT := 16#0000,
            P := 38,
            OUT => "DELTA D"."MAX TEMP",
            ENO => #_w8);
   IF #_w8 THEN
       VAL_STRG(IN := "DELTA D"."MAX T4",
                SIZE := 5,
                PREC := 1,
                FORMAT := 16#0000,
                P := 46,
                OUT => "DELTA D"."MAX TEMP");
   END_IF;
   VAL_STRG(IN := "DELTA D".F1,
            SIZE := 5,
            PREC := 2,
            FORMAT := 16#0000,
            P := 17,
            OUT => "DELTA D"."F ZERO",
            ENO => #_w9);
   VAL_STRG(EN := #_w9,
            IN := "DELTA D".F2,
            SIZE := 5,
            PREC := 2,
            FORMAT := 16#0000,
            P := 24,
            OUT => "DELTA D"."F ZERO",
            ENO => #_w10);
   VAL_STRG(EN := #_w10,
            IN := "DELTA D".F3,
            SIZE := 5,
            PREC := 2,
            FORMAT := 16#0000,
            P := 31,
            OUT => "DELTA D"."F ZERO",
            ENO => #_w11);
   VAL_STRG(EN := #_w11,
            IN := "DELTA D".F4,
            SIZE := 5,
            PREC := 2,
            FORMAT := 16#0000,
            P := 38,
            OUT => "DELTA D"."F ZERO",
            ENO => #_w12);
   IF #_w12 THEN
       VAL_STRG(IN := "DELTA D".F5, SIZE := 5, PREC := 2, FORMAT := 16#0000, P := 46, OUT => "DELTA D"."F ZERO");
   END_IF;
   VAL_STRG(IN := "DELTA D".F0, SIZE := 5, PREC := 2, FORMAT := 16#0000, P := 52, OUT => "DELTA D"."MIN F0");
END_REGION

REGION Network 19
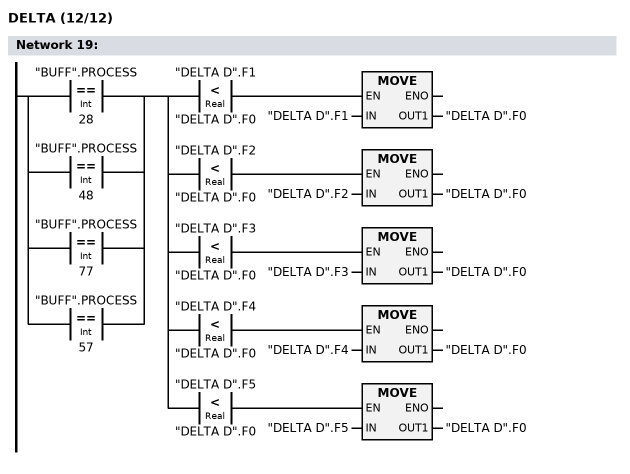
   RUNG wire#powerrail
      { S7_Templates := "SrcType := Int" } EQ_Contact(in1 := "BUFF".PROCESS, in2 := 28)
      wire#w1
      { S7_Templates := "SrcType := Real" } LT_Contact(in1 := "DELTA D".F1, in2 := "DELTA D".F0)
      Move(in := "DELTA D".F1, out1 => "DELTA D".F0)
   END_RUNG
   RUNG wire#powerrail
      { S7_Templates := "SrcType := Int" } EQ_Contact(in1 := "BUFF".PROCESS, in2 := 48)
   END_RUNG wire#w1
   RUNG wire#powerrail
      { S7_Templates := "SrcType := Int" } EQ_Contact(in1 := "BUFF".PROCESS, in2 := 77)
   END_RUNG wire#w1
   RUNG wire#powerrail
      { S7_Templates := "SrcType := Int" } EQ_Contact(in1 := "BUFF".PROCESS, in2 := 57)
   END_RUNG wire#w1
   RUNG wire#w1
      { S7_Templates := "SrcType := Real" } LT_Contact(in1 := "DELTA D".F2, in2 := "DELTA D".F0)
      Move(in := "DELTA D".F2, out1 => "DELTA D".F0)
   END_RUNG
   RUNG wire#w1
      { S7_Templates := "SrcType := Real" } LT_Contact(in1 := "DELTA D".F3, in2 := "DELTA D".F0)
      Move(in := "DELTA D".F3, out1 => "DELTA D".F0)
   END_RUNG
   RUNG wire#w1
      { S7_Templates := "SrcType := Real" } LT_Contact(in1 := "DELTA D".F4, in2 := "DELTA D".F0)
      Move(in := "DELTA D".F4, out1 => "DELTA D".F0)
   END_RUNG
   RUNG wire#w1
      { S7_Templates := "SrcType := Real" } LT_Contact(in1 := "DELTA D".F5, in2 := "DELTA D".F0)
      Move(in := "DELTA D".F5, out1 => "DELTA D".F0)
   END_RUNG
   // the same network as SCL:
   #_w1 := ("BUFF".PROCESS = 28) OR ("BUFF".PROCESS = 48) OR ("BUFF".PROCESS = 77) OR ("BUFF".PROCESS = 57);
   IF #_w1 AND ("DELTA D".F1 < "DELTA D".F0) THEN "DELTA D".F0 := "DELTA D".F1; END_IF;
   IF #_w1 AND ("DELTA D".F2 < "DELTA D".F0) THEN "DELTA D".F0 := "DELTA D".F2; END_IF;
   IF #_w1 AND ("DELTA D".F3 < "DELTA D".F0) THEN "DELTA D".F0 := "DELTA D".F3; END_IF;
   IF #_w1 AND ("DELTA D".F4 < "DELTA D".F0) THEN "DELTA D".F0 := "DELTA D".F4; END_IF;
   IF #_w1 AND ("DELTA D".F5 < "DELTA D".F0) THEN "DELTA D".F0 := "DELTA D".F5; END_IF;
END_REGION
END_FUNCTION

FUNCTION "END PRINT" : Void   // FC19, LAD
{ S7_Optimized_Access := 'TRUE' }
// stored: SetENOAutomatically false
BEGIN

REGION Network 1: RECORD TIME
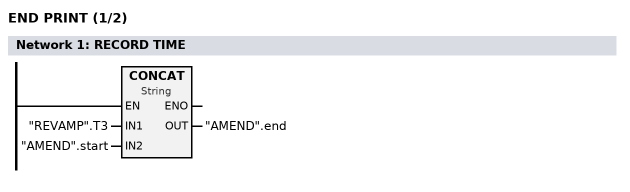
   RUNG wire#powerrail
      { S7_Templates := "[card := 2, str_type := String]" } CONCAT(IN1 := "REVAMP".T3, IN2 := "AMEND".start, OUT => "AMEND".end)
   END_RUNG
   // the same network as SCL:
   CONCAT(IN1 := "REVAMP".T3, IN2 := "AMEND".start, OUT => "AMEND".end);
END_REGION

REGION Network 2: PV CONCATE
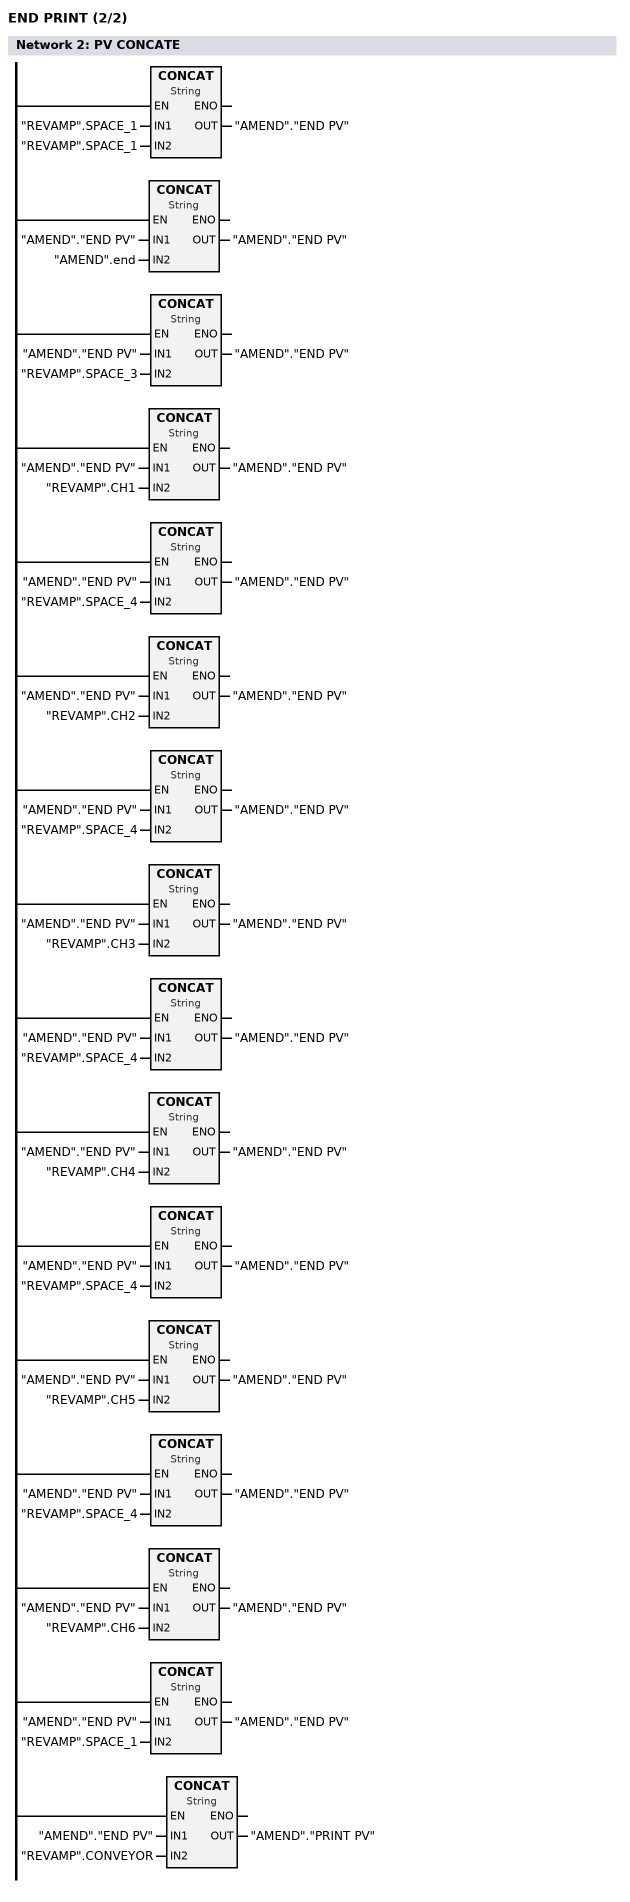
   RUNG wire#powerrail
      { S7_Templates := "[card := 2, str_type := String]" } CONCAT(IN1 := "REVAMP".SPACE_1, IN2 := "REVAMP".SPACE_1, OUT => "AMEND"."END PV")
   END_RUNG
   RUNG wire#powerrail
      { S7_Templates := "[card := 2, str_type := String]" } CONCAT(IN1 := "AMEND"."END PV", IN2 := "AMEND".end, OUT => "AMEND"."END PV")
   END_RUNG
   RUNG wire#powerrail
      { S7_Templates := "[card := 2, str_type := String]" } CONCAT(IN1 := "AMEND"."END PV", IN2 := "REVAMP".SPACE_3, OUT => "AMEND"."END PV")
   END_RUNG
   RUNG wire#powerrail
      { S7_Templates := "[card := 2, str_type := String]" } CONCAT(IN1 := "AMEND"."END PV", IN2 := "REVAMP".CH1, OUT => "AMEND"."END PV")
   END_RUNG
   RUNG wire#powerrail
      { S7_Templates := "[card := 2, str_type := String]" } CONCAT(IN1 := "AMEND"."END PV", IN2 := "REVAMP".SPACE_4, OUT => "AMEND"."END PV")
   END_RUNG
   RUNG wire#powerrail
      { S7_Templates := "[card := 2, str_type := String]" } CONCAT(IN1 := "AMEND"."END PV", IN2 := "REVAMP".CH2, OUT => "AMEND"."END PV")
   END_RUNG
   RUNG wire#powerrail
      { S7_Templates := "[card := 2, str_type := String]" } CONCAT(IN1 := "AMEND"."END PV", IN2 := "REVAMP".SPACE_4, OUT => "AMEND"."END PV")
   END_RUNG
   RUNG wire#powerrail
      { S7_Templates := "[card := 2, str_type := String]" } CONCAT(IN1 := "AMEND"."END PV", IN2 := "REVAMP".CH3, OUT => "AMEND"."END PV")
   END_RUNG
   RUNG wire#powerrail
      { S7_Templates := "[card := 2, str_type := String]" } CONCAT(IN1 := "AMEND"."END PV", IN2 := "REVAMP".SPACE_4, OUT => "AMEND"."END PV")
   END_RUNG
   RUNG wire#powerrail
      { S7_Templates := "[card := 2, str_type := String]" } CONCAT(IN1 := "AMEND"."END PV", IN2 := "REVAMP".CH4, OUT => "AMEND"."END PV")
   END_RUNG
   RUNG wire#powerrail
      { S7_Templates := "[card := 2, str_type := String]" } CONCAT(IN1 := "AMEND"."END PV", IN2 := "REVAMP".SPACE_4, OUT => "AMEND"."END PV")
   END_RUNG
   RUNG wire#powerrail
      { S7_Templates := "[card := 2, str_type := String]" } CONCAT(IN1 := "AMEND"."END PV", IN2 := "REVAMP".CH5, OUT => "AMEND"."END PV")
   END_RUNG
   RUNG wire#powerrail
      { S7_Templates := "[card := 2, str_type := String]" } CONCAT(IN1 := "AMEND"."END PV", IN2 := "REVAMP".SPACE_4, OUT => "AMEND"."END PV")
   END_RUNG
   RUNG wire#powerrail
      { S7_Templates := "[card := 2, str_type := String]" } CONCAT(IN1 := "AMEND"."END PV", IN2 := "REVAMP".CH6, OUT => "AMEND"."END PV")
   END_RUNG
   RUNG wire#powerrail
      { S7_Templates := "[card := 2, str_type := String]" } CONCAT(IN1 := "AMEND"."END PV", IN2 := "REVAMP".SPACE_1, OUT => "AMEND"."END PV")
   END_RUNG
   RUNG wire#powerrail
      { S7_Templates := "[card := 2, str_type := String]" } CONCAT(IN1 := "AMEND"."END PV", IN2 := "REVAMP".CONVEYOR, OUT => "AMEND"."PRINT PV")
   END_RUNG
   // the same network as SCL:
   CONCAT(IN1 := "REVAMP".SPACE_1, IN2 := "REVAMP".SPACE_1, OUT => "AMEND"."END PV");
   CONCAT(IN1 := "AMEND"."END PV", IN2 := "AMEND".end, OUT => "AMEND"."END PV");
   CONCAT(IN1 := "AMEND"."END PV", IN2 := "REVAMP".SPACE_3, OUT => "AMEND"."END PV");
   CONCAT(IN1 := "AMEND"."END PV", IN2 := "REVAMP".CH1, OUT => "AMEND"."END PV");
   CONCAT(IN1 := "AMEND"."END PV", IN2 := "REVAMP".SPACE_4, OUT => "AMEND"."END PV");
   CONCAT(IN1 := "AMEND"."END PV", IN2 := "REVAMP".CH2, OUT => "AMEND"."END PV");
   CONCAT(IN1 := "AMEND"."END PV", IN2 := "REVAMP".SPACE_4, OUT => "AMEND"."END PV");
   CONCAT(IN1 := "AMEND"."END PV", IN2 := "REVAMP".CH3, OUT => "AMEND"."END PV");
   CONCAT(IN1 := "AMEND"."END PV", IN2 := "REVAMP".SPACE_4, OUT => "AMEND"."END PV");
   CONCAT(IN1 := "AMEND"."END PV", IN2 := "REVAMP".CH4, OUT => "AMEND"."END PV");
   CONCAT(IN1 := "AMEND"."END PV", IN2 := "REVAMP".SPACE_4, OUT => "AMEND"."END PV");
   CONCAT(IN1 := "AMEND"."END PV", IN2 := "REVAMP".CH5, OUT => "AMEND"."END PV");
   CONCAT(IN1 := "AMEND"."END PV", IN2 := "REVAMP".SPACE_4, OUT => "AMEND"."END PV");
   CONCAT(IN1 := "AMEND"."END PV", IN2 := "REVAMP".CH6, OUT => "AMEND"."END PV");
   CONCAT(IN1 := "AMEND"."END PV", IN2 := "REVAMP".SPACE_1, OUT => "AMEND"."END PV");
   CONCAT(IN1 := "AMEND"."END PV", IN2 := "REVAMP".CONVEYOR, OUT => "AMEND"."PRINT PV");
END_REGION
END_FUNCTION

FUNCTION "ampoule" : Void   // FC6, LAD
{ S7_Optimized_Access := 'TRUE' }
// stored: SetENOAutomatically false
   VAR_TEMP   // added for the SCL form of the ladder/FBD networks
      _w1 : Bool;
      _w2 : Bool;
   END_VAR
BEGIN

REGION Network 1
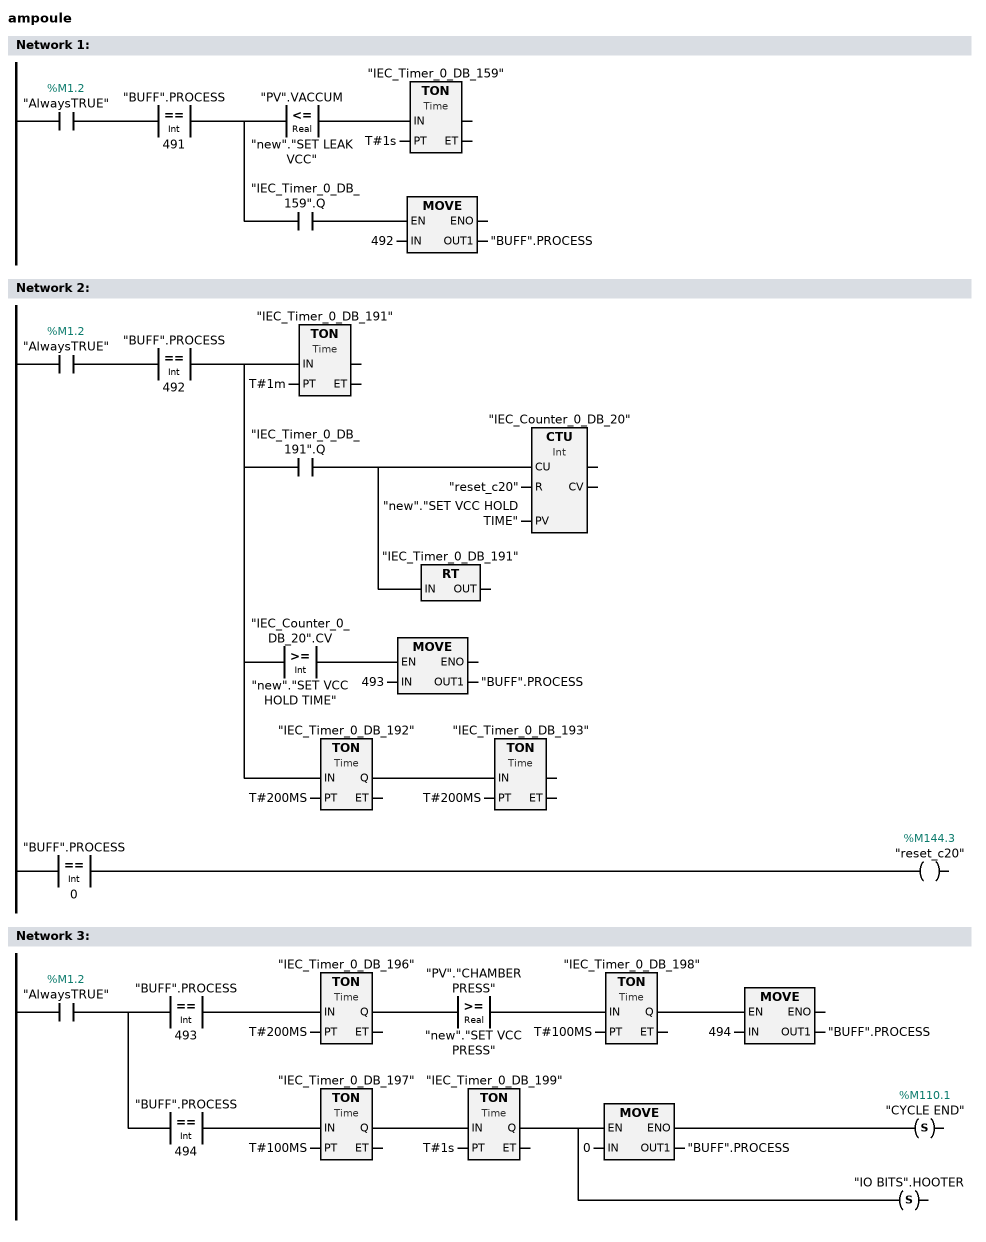
   RUNG wire#powerrail
      Contact( "AlwaysTRUE" )
      { S7_Templates := "SrcType := Int" } EQ_Contact(in1 := "BUFF".PROCESS, in2 := 491)
      wire#w1
      { S7_Templates := "SrcType := Real" } LE_Contact(in1 := "PV".VACCUM, in2 := "new"."SET LEAK VCC")
      { S7_Templates := "time_type := Time" } "IEC_Timer_0_DB_159".TON(pt := T#1s, et =>)
   END_RUNG
   RUNG wire#w1
      Contact( "IEC_Timer_0_DB_159".Q )
      Move(in := 492, out1 => "BUFF".PROCESS)
   END_RUNG
   // the same network as SCL:
   #_w1 := "AlwaysTRUE" AND ("BUFF".PROCESS = 491);
   "IEC_Timer_0_DB_159".TON(IN := #_w1 AND ("PV".VACCUM <= "new"."SET LEAK VCC"), PT := T#1s);
   IF #_w1 AND "IEC_Timer_0_DB_159".Q THEN "BUFF".PROCESS := 492; END_IF;
END_REGION

REGION Network 2
   RUNG wire#powerrail
      Contact( "AlwaysTRUE" )
      { S7_Templates := "SrcType := Int" } EQ_Contact(in1 := "BUFF".PROCESS, in2 := 492)
      wire#w1
      { S7_Templates := "time_type := Time" } "IEC_Timer_0_DB_191".TON(pt := T#1m, et =>)
   END_RUNG
   RUNG wire#w1
      Contact( "IEC_Timer_0_DB_191".Q )
      wire#w2
      { S7_Templates := "value_type := Int" } "IEC_Counter_0_DB_20".CTU(r := "reset_c20", pv := "new"."SET VCC HOLD TIME", cv =>)
   END_RUNG
   RUNG wire#w2
      RT_Coil( "IEC_Timer_0_DB_191" )
   END_RUNG
   RUNG wire#w1
      { S7_Templates := "SrcType := Int" } GE_Contact(in1 := "IEC_Counter_0_DB_20".CV, in2 := "new"."SET VCC HOLD TIME")
      Move(in := 493, out1 => "BUFF".PROCESS)
   END_RUNG
   RUNG wire#w1
      { S7_Templates := "time_type := Time" } "IEC_Timer_0_DB_192".TON(pt := T#200MS, et =>)
      { S7_Templates := "time_type := Time" } "IEC_Timer_0_DB_193".TON(pt := T#200MS, et =>)
   END_RUNG
   RUNG wire#powerrail
      { S7_Templates := "SrcType := Int" } EQ_Contact(in1 := "BUFF".PROCESS, in2 := 0)
      Coil( "reset_c20" )
   END_RUNG
   // the same network as SCL:
   #_w1 := "AlwaysTRUE" AND ("BUFF".PROCESS = 492);
   "IEC_Timer_0_DB_191".TON(IN := #_w1, PT := T#1m);
   #_w2 := #_w1 AND "IEC_Timer_0_DB_191".Q;
   "IEC_Counter_0_DB_20".CTU(CU := #_w2, R := "reset_c20", PV := "new"."SET VCC HOLD TIME");
   IF #_w2 THEN RESET_TIMER("IEC_Timer_0_DB_191"); END_IF;
   IF #_w1 AND ("IEC_Counter_0_DB_20".CV >= "new"."SET VCC HOLD TIME") THEN "BUFF".PROCESS := 493; END_IF;
   "IEC_Timer_0_DB_192".TON(IN := #_w1, PT := T#200MS);
   "IEC_Timer_0_DB_193".TON(IN := "IEC_Timer_0_DB_192".Q, PT := T#200MS);
   "reset_c20" := "BUFF".PROCESS = 0;
END_REGION

REGION Network 3
   RUNG wire#powerrail
      Contact( "AlwaysTRUE" )
      wire#w1
      { S7_Templates := "SrcType := Int" } EQ_Contact(in1 := "BUFF".PROCESS, in2 := 493)
      { S7_Templates := "time_type := Time" } "IEC_Timer_0_DB_196".TON(pt := T#200MS, et =>)
      { S7_Templates := "SrcType := Real" } GE_Contact(in1 := "PV"."CHAMBER PRESS", in2 := "new"."SET VCC PRESS")
      { S7_Templates := "time_type := Time" } "IEC_Timer_0_DB_198".TON(pt := T#100MS, et =>)
      Move(in := 494, out1 => "BUFF".PROCESS)
   END_RUNG
   RUNG wire#w1
      { S7_Templates := "SrcType := Int" } EQ_Contact(in1 := "BUFF".PROCESS, in2 := 494)
      { S7_Templates := "time_type := Time" } "IEC_Timer_0_DB_197".TON(pt := T#100MS, et =>)
      { S7_Templates := "time_type := Time" } "IEC_Timer_0_DB_199".TON(pt := T#1s, et =>)
      wire#w2
      Move(in := 0, out1 => "BUFF".PROCESS)
      S_Coil( "CYCLE END" )
   END_RUNG
   RUNG wire#w2
      S_Coil( "IO BITS".HOOTER )
   END_RUNG
   // the same network as SCL:
   "IEC_Timer_0_DB_196".TON(IN := "AlwaysTRUE" AND ("BUFF".PROCESS = 493), PT := T#200MS);
   "IEC_Timer_0_DB_198".TON(IN := "IEC_Timer_0_DB_196".Q AND ("PV"."CHAMBER PRESS" >= "new"."SET VCC PRESS"),
                           PT := T#100MS);
   IF "IEC_Timer_0_DB_198".Q THEN "BUFF".PROCESS := 494; END_IF;
   "IEC_Timer_0_DB_197".TON(IN := "AlwaysTRUE" AND ("BUFF".PROCESS = 494), PT := T#100MS);
   "IEC_Timer_0_DB_199".TON(IN := "IEC_Timer_0_DB_197".Q, PT := T#1s);
   IF "IEC_Timer_0_DB_199".Q THEN
       "BUFF".PROCESS := 0;
       "CYCLE END" := TRUE;
       "IO BITS".HOOTER := TRUE;
   END_IF;
END_REGION
END_FUNCTION

FUNCTION_BLOCK "DATALOG TRIGGER BLOCK"   // FB11, LAD
{ S7_Optimized_Access := 'TRUE' }
// stored: MemoryReserve 100, SetENOAutomatically false
   VAR_INPUT
      "SET TIME" : Int;
      RESET : Bool;
      INPUT : Bool;
   END_VAR
   VAR_OUTPUT
      "PRESENT VALUE OF TIME" : Int;
      SEC : Int;
      DONE : Bool;
      "TRIGGER BIT" : Bool;
      "ALARM BIT" : Bool;
   END_VAR
   VAR
      "TIMER 1" { S7_SetPoint := 'True'} : IEC_TIMER;
   END_VAR
   VAR RETAIN
      "COUNTER1 0" { S7_SetPoint := 'True'} : IEC_COUNTER;
      "COUNTER1 1" { S7_SetPoint := 'True'} : IEC_COUNTER;
      TPULSE { S7_SetPoint := 'True'} : IEC_TIMER;
   END_VAR
   VAR_TEMP   // added for the SCL form of the ladder/FBD networks
      _w1 : Bool;
      _w2 : Bool;
   END_VAR
BEGIN

REGION Network 2
